KUKA KRL program: EPS_2_26115_SA7007_A_20260219035546.src

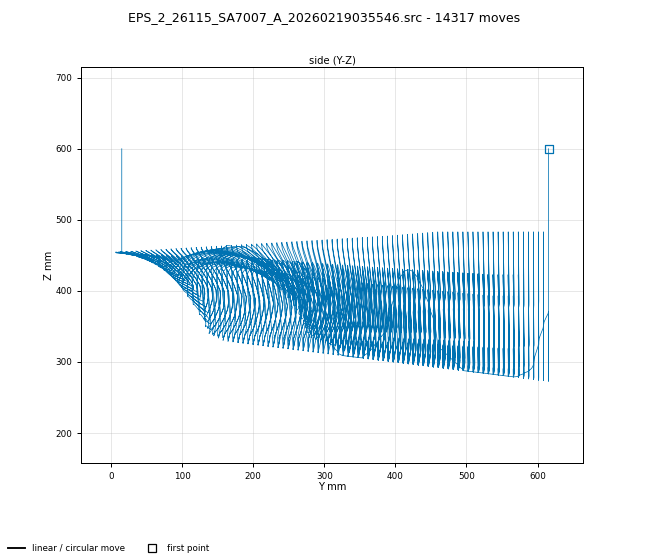
[picture p0: tool path of EPS_2_26115_SA7007_A_20260219035546.src, 14317 of 14319 moves have a stored position in this frame; points joined in program order, loops and branches not executed]
&ACCESS RVP
&REL 4
&COMMENT QRS 19112012
&PARAM EDITMASK = *
DEF PART()
EXT BAS (BAS_COMMAND :IN,REAL :IN )
INT I
BAS (#INITMOV,0 )

;KUKA QRS Post kuka4.cps  Date:22-06-2017 !

File_ID=3063

QRS_PRE_INIT()

;Init var - Until changes are made in qrs_pre_init
Outlet_Square_prg=0
Inlet_1_Square_prg=0
Inlet_2_Square_prg=0
Inlet_3_Square_prg=0
Inlet_4_Square_prg=0
Inlet_5_Square_prg=0

Outlet_1={X 0.000, Y 460.000, Z 382.500, B 0.000, E1 0.000 }
Inlet_1={X 0.000, Y 532.890, Z 292.500, B 0.000, E1 90.000 }
Inlet_2={X 0.000, Y 530.720, Z 322.500, B 0.000, E1 180.000 }
Inlet_3={X 0.000, Y 530.720, Z 322.500, B 0.000, E1 270.000 }
Outlet_1_type=201
Inlet_1_type=201
Inlet_2_type=201
Inlet_3_type=201
;QRS#1=Sidecore dimensions
;QRS#2=200-8" PVC SDR 35 Cut Back
;QRS#3=200-8" PVC SDR 35
;QRS#4=200-8" PVC SDR 35
;QRS#5=200-8" PVC SDR 35
;QRS#6=
;QRS#7=
;QRS#8=
;QRS#9=12-08 PSX
;QRS#10=12-08 PSX
;QRS#11=12-08 PSX
;QRS#12=12-08 PSX
;QRS#13=
;QRS#14=
;QRS#15=
;QRS#16=1220x127x762 2,5'
;QRS#17=EPS Height
;QRS#18=483
;QRS#19=*
;QRS#20= UPDATED VERSION 22-06-2017
;QRS#21=*
Outlet_Square=0100
Inlet_1_Square=0100
Inlet_2_Square=0100
Inlet_3_Square=0100
Inlet_4_Square=0
Inlet_5_Square=0
Mill_Square=1
Outlet_Square_Prg=214
Inlet_1_Square_prg=204
Inlet_2_Square_prg=204
Inlet_3_Square_prg=204

QRS_INIT()

$ADVANCE=5

; T1
PTP {E1 173.498,E2 173.498}
PTP {X 0,Y 615.498,A -85,B 0,C 180,E1 173.498,E2 173.498,E3 0,E4 0,E5 0,E6 0}
QRS_SPEED_INIT()
LIN {X 0,Y 615.498,Z 600,A -85,B 0,C 180,E1 173.498,E2 173.498,E3 0,E4 0,E5 0,E6 0} C_VEL
LIN {X 0,Y 615.498,Z 383.731,A -85,B 0,C 180,E1 173.498,E2 173.498} C_VEL
LIN {X 0,Y 615.498,Z 372.852,A -85,B 0,C 180,E1 173.498,E2 173.498} C_VEL
LIN {X 0,Y 615.496,Z 371.208,A -85,B 0,C 180,E1 173.418,E2 173.418} C_VEL
LIN {X 0,Y 615.497,Z 363.536,A -85,B 0,C 180,E1 172.455,E2 172.455} C_VEL
LIN {X 0,Y 615.498,Z 353.758,A -85,B 0,C 180,E1 171.463,E2 171.463} C_VEL
LIN {X 0,Y 615.498,Z 343.492,A -85,B 0,C 180,E1 170.636,E2 170.636} C_VEL
LIN {X 0,Y 615.458,Z 331.934,A -85,B 0,C 180,E1 169.888,E2 169.888} C_VEL
LIN {X 0,Y 615.433,Z 320.391,A -85,B 0,C 180,E1 169.305,E2 169.305} C_VEL
LIN {X 0,Y 615.457,Z 308.449,A -85,B 0,C 180,E1 168.848,E2 168.848} C_VEL
LIN {X 0,Y 615.487,Z 296.38,A -85,B 0,C 180,E1 168.515,E2 168.515} C_VEL
LIN {X 0,Y 615.495,Z 289.406,A -85,B 0,C 180,E1 168.369,E2 168.369} C_VEL
LIN {X 0,Y 615.472,Z 286.424,A -85,B 0,C 180,E1 166.075,E2 166.075} C_VEL
LIN {X 0,Y 615.45,Z 282.996,A -85,B 0,C 180,E1 163.412,E2 163.412} C_VEL
LIN {X 0,Y 615.494,Z 279.512,A -85,B 0,C 180,E1 160.662,E2 160.662} C_VEL
LIN {X 0,Y 615.46,Z 276.011,A -85,B 0,C 180,E1 157.862,E2 157.862} C_VEL
LIN {X 0,Y 615.467,Z 273.391,A -85,B 0,C 180,E1 155.727,E2 155.727} C_VEL
LIN {X 0,Y 615.489,Z 272.693,A -85,B 0,C 180,E1 155.008,E2 155.008} C_VEL
LIN {X 0,Y 615.468,Z 272.69,A -85,B 0,C 180,E1 152.084,E2 152.084} C_VEL
LIN {X 0,Y 615.473,Z 272.695,A -85,B 0,C 180,E1 149.839,E2 149.839} C_VEL
LIN {X 0,Y 615.495,Z 272.7,A -85,B 0,C 180,E1 147.543,E2 147.543} C_VEL
LIN {X 0,Y 615.482,Z 272.69,A -85,B 0,C 180,E1 145.184,E2 145.184} C_VEL
LIN {X 0,Y 615.492,Z 272.682,A -85,B 0,C 180,E1 142.758,E2 142.758} C_VEL
LIN {X 0,Y 615.496,Z 272.7,A -85,B 0,C 180,E1 139.91,E2 139.91} C_VEL
LIN {X 0,Y 615.488,Z 272.683,A -85,B 0,C 180,E1 136.953,E2 136.953} C_VEL
LIN {X 0,Y 615.489,Z 272.698,A -85,B 0,C 180,E1 133.997,E2 133.997} C_VEL
LIN {X 0,Y 615.487,Z 272.684,A -85,B 0,C 180,E1 131.094,E2 131.094} C_VEL
LIN {X 0,Y 615.488,Z 272.687,A -85,B 0,C 180,E1 128.905,E2 128.905} C_VEL
LIN {X 0,Y 615.484,Z 272.704,A -85,B 0,C 180,E1 126.425,E2 126.425} C_VEL
LIN {X 0,Y 615.49,Z 272.727,A -85,B 0,C 180,E1 124.701,E2 124.701} C_VEL
LIN {X 0,Y 615.482,Z 277.506,A -85,B 0,C 180,E1 122.329,E2 122.329} C_VEL
LIN {X 0,Y 615.472,Z 282.453,A -85,B 0,C 180,E1 119.791,E2 119.791} C_VEL
LIN {X 0,Y 615.46,Z 287.533,A -85,B 0,C 180,E1 117.039,E2 117.039} C_VEL
LIN {X 0,Y 615.461,Z 291.397,A -85,B 0,C 180,E1 114.993,E2 114.993} C_VEL
LIN {X 0,Y 615.482,Z 296.491,A -85,B 0,C 180,E1 112.344,E2 112.344} C_VEL
LIN {X 0,Y 615.482,Z 301.009,A -85,B 0,C 180,E1 110.033,E2 110.033} C_VEL
LIN {X 0,Y 615.484,Z 306.513,A -85,B 0,C 180,E1 107.271,E2 107.271} C_VEL
LIN {X 0,Y 615.467,Z 311.996,A -85,B 0,C 180,E1 104.55,E2 104.55} C_VEL
LIN {X 0,Y 615.479,Z 317.495,A -85,B 0,C 180,E1 101.861,E2 101.861} C_VEL
LIN {X 0,Y 615.496,Z 318.09,A -85,B 0,C 180,E1 101.568,E2 101.568} C_VEL
LIN {X 0,Y 615.485,Z 332.738,A -85,B 0,C 180,E1 101.235,E2 101.235} C_VEL
LIN {X 0,Y 615.452,Z 345.032,A -85,B 0,C 180,E1 100.827,E2 100.827} C_VEL
LIN {X 0,Y 615.452,Z 357.201,A -85,B 0,C 180,E1 100.278,E2 100.278} C_VEL
LIN {X 0,Y 615.496,Z 368.575,A -85,B 0,C 180,E1 99.613,E2 99.613} C_VEL
LIN {X 0,Y 615.498,Z 378.822,A -85,B 0,C 180,E1 98.867,E2 98.867} C_VEL
LIN {X 0,Y 615.498,Z 388.033,A -85,B 0,C 180,E1 98.041,E2 98.041} C_VEL
LIN {X 0,Y 615.499,Z 396.892,A -85,B 0,C 180,E1 97.057,E2 97.057} C_VEL
LIN {X 0,Y 615.497,Z 404.123,A -85,B 0,C 180,E1 96.063,E2 96.063} C_VEL
LIN {X 0,Y 615.497,Z 408.958,A -85,B 0,C 180,E1 95.241,E2 95.241} C_VEL
LIN {X 0,Y 615.494,Z 413.658,A -85,B 0,C 180,E1 94.256,E2 94.256} C_VEL
LIN {X 0,Y 615.494,Z 417.254,A -85,B 0,C 180,E1 93.273,E2 93.273} C_VEL
LIN {X 0,Y 615.496,Z 419.115,A -85,B 0,C 180,E1 92.618,E2 92.618} C_VEL
LIN {X 0,Y 615.5,Z 420.533,A -85,B 0,C 180,E1 91.963,E2 91.963} C_VEL
LIN {X 0,Y 615.496,Z 422.141,A -85,B 0,C 180,E1 90.654,E2 90.654} C_VEL
LIN {X 0,Y 615.495,Z 422.384,A -85,B 0,C 180,E1 90,E2 90} C_VEL
LIN {X 0,Y 615.495,Z 422.206,A -85,B 0,C 180,E1 89.346,E2 89.346} C_VEL
LIN {X 0,Y 615.5,Z 420.682,A -85,B 0,C 180,E1 88.037,E2 88.037} C_VEL
LIN {X 0,Y 615.498,Z 419.341,A -85,B 0,C 180,E1 87.382,E2 87.382} C_VEL
LIN {X 0,Y 615.496,Z 416.494,A -85,B 0,C 180,E1 86.399,E2 86.399} C_VEL
LIN {X 0,Y 615.498,Z 412.634,A -85,B 0,C 180,E1 85.416,E2 85.416} C_VEL
LIN {X 0,Y 615.498,Z 407.651,A -85,B 0,C 180,E1 84.43,E2 84.43} C_VEL
LIN {X 0,Y 615.496,Z 401.208,A -85,B 0,C 180,E1 83.418,E2 83.418} C_VEL
LIN {X 0,Y 615.497,Z 393.536,A -85,B 0,C 180,E1 82.455,E2 82.455} C_VEL
LIN {X 0,Y 615.498,Z 383.758,A -85,B 0,C 180,E1 81.463,E2 81.463} C_VEL
LIN {X 0,Y 615.498,Z 373.492,A -85,B 0,C 180,E1 80.636,E2 80.636} C_VEL
LIN {X 0,Y 615.46,Z 361.934,A -85,B 0,C 180,E1 79.888,E2 79.888} C_VEL
LIN {X 0,Y 615.439,Z 350.346,A -85,B 0,C 180,E1 79.303,E2 79.303} C_VEL
LIN {X 0,Y 615.467,Z 338.434,A -85,B 0,C 180,E1 78.848,E2 78.848} C_VEL
LIN {X 0,Y 615.494,Z 326.38,A -85,B 0,C 180,E1 78.515,E2 78.515} C_VEL
LIN {X 0,Y 615.497,Z 318.103,A -85,B 0,C 180,E1 78.348,E2 78.348} C_VEL
LIN {X 0,Y 615.476,Z 313.45,A -85,B 0,C 180,E1 76.073,E2 76.073} C_VEL
LIN {X 0,Y 615.476,Z 308.058,A -85,B 0,C 180,E1 73.413,E2 73.413} C_VEL
LIN {X 0,Y 615.486,Z 302.567,A -85,B 0,C 180,E1 70.662,E2 70.662} C_VEL
LIN {X 0,Y 615.487,Z 297.064,A -85,B 0,C 180,E1 67.863,E2 67.863} C_VEL
LIN {X 0,Y 615.483,Z 292.945,A -85,B 0,C 180,E1 65.728,E2 65.728} C_VEL
LIN {X 0,Y 615.456,Z 288.826,A -85,B 0,C 180,E1 63.554,E2 63.554} C_VEL
LIN {X 0,Y 615.441,Z 284.694,A -85,B 0,C 180,E1 61.339,E2 61.339} C_VEL
LIN {X 0,Y 615.495,Z 280.115,A -85,B 0,C 180,E1 58.913,E2 58.913} C_VEL
LIN {X 0,Y 615.481,Z 275.287,A -85,B 0,C 180,E1 56.467,E2 56.467} C_VEL
LIN {X 0,Y 615.491,Z 272.697,A -85,B 0,C 180,E1 55.185,E2 55.185} C_VEL
LIN {X 0,Y 615.489,Z 272.701,A -85,B 0,C 180,E1 52.758,E2 52.758} C_VEL
LIN {X 0,Y 615.472,Z 272.7,A -85,B 0,C 180,E1 49.913,E2 49.913} C_VEL
LIN {X 0,Y 615.492,Z 272.693,A -85,B 0,C 180,E1 46.953,E2 46.953} C_VEL
LIN {X 0,Y 615.466,Z 272.7,A -85,B 0,C 180,E1 44.152,E2 44.152} C_VEL
LIN {X 0,Y 615.469,Z 272.7,A -85,B 0,C 180,E1 41.476,E2 41.476} C_VEL
LIN {X 0,Y 615.492,Z 272.694,A -85,B 0,C 180,E1 38.904,E2 38.904} C_VEL
LIN {X 0,Y 615.464,Z 272.7,A -85,B 0,C 180,E1 36.427,E2 36.427} C_VEL
LIN {X 0,Y 615.489,Z 272.727,A -85,B 0,C 180,E1 34.815,E2 34.815} C_VEL
LIN {X 0,Y 615.484,Z 277.586,A -85,B 0,C 180,E1 32.33,E2 32.33} C_VEL
LIN {X 0,Y 615.471,Z 282.454,A -85,B 0,C 180,E1 29.791,E2 29.791} C_VEL
LIN {X 0,Y 615.459,Z 287.533,A -85,B 0,C 180,E1 27.039,E2 27.039} C_VEL
LIN {X 0,Y 615.461,Z 291.397,A -85,B 0,C 180,E1 24.993,E2 24.993} C_VEL
LIN {X 0,Y 615.482,Z 296.491,A -85,B 0,C 180,E1 22.344,E2 22.344} C_VEL
LIN {X 0,Y 615.482,Z 301.009,A -85,B 0,C 180,E1 20.033,E2 20.033} C_VEL
LIN {X 0,Y 615.485,Z 306.513,A -85,B 0,C 180,E1 17.271,E2 17.271} C_VEL
LIN {X 0,Y 615.468,Z 311.996,A -85,B 0,C 180,E1 14.55,E2 14.55} C_VEL
LIN {X 0,Y 615.479,Z 317.495,A -85,B 0,C 180,E1 11.861,E2 11.861} C_VEL
LIN {X 0,Y 615.496,Z 318.09,A -85,B 0,C 180,E1 11.568,E2 11.568} C_VEL
LIN {X 0,Y 615.485,Z 332.737,A -85,B 0,C 180,E1 11.235,E2 11.235} C_VEL
LIN {X 0,Y 615.452,Z 345.032,A -85,B 0,C 180,E1 10.827,E2 10.827} C_VEL
LIN {X 0,Y 615.452,Z 357.2,A -85,B 0,C 180,E1 10.278,E2 10.278} C_VEL
LIN {X 0,Y 615.496,Z 368.574,A -85,B 0,C 180,E1 9.613,E2 9.613} C_VEL
LIN {X 0,Y 615.498,Z 378.822,A -85,B 0,C 180,E1 8.867,E2 8.867} C_VEL
LIN {X 0,Y 615.498,Z 388.033,A -85,B 0,C 180,E1 8.041,E2 8.041} C_VEL
LIN {X 0,Y 615.499,Z 396.891,A -85,B 0,C 180,E1 7.057,E2 7.057} C_VEL
LIN {X 0,Y 615.497,Z 404.123,A -85,B 0,C 180,E1 6.063,E2 6.063} C_VEL
LIN {X 0,Y 615.497,Z 408.958,A -85,B 0,C 180,E1 5.241,E2 5.241} C_VEL
LIN {X 0,Y 615.494,Z 413.658,A -85,B 0,C 180,E1 4.256,E2 4.256} C_VEL
LIN {X 0,Y 615.494,Z 417.254,A -85,B 0,C 180,E1 3.273,E2 3.273} C_VEL
LIN {X 0,Y 615.496,Z 419.115,A -85,B 0,C 180,E1 2.618,E2 2.618} C_VEL
LIN {X 0,Y 615.5,Z 420.533,A -85,B 0,C 180,E1 1.963,E2 1.963} C_VEL
LIN {X 0,Y 615.496,Z 422.141,A -85,B 0,C 180,E1 0.654,E2 0.654} C_VEL
LIN {X 0,Y 615.495,Z 422.384,A -85,B 0,C 180,E1 0,E2 0} C_VEL
LIN {X 0,Y 615.495,Z 422.206,A -85,B 0,C 180,E1 -0.654,E2 -0.654} C_VEL
LIN {X 0,Y 615.5,Z 420.682,A -85,B 0,C 180,E1 -1.963,E2 -1.963} C_VEL
LIN {X 0,Y 615.498,Z 419.341,A -85,B 0,C 180,E1 -2.618,E2 -2.618} C_VEL
LIN {X 0,Y 615.496,Z 416.494,A -85,B 0,C 180,E1 -3.601,E2 -3.601} C_VEL
LIN {X 0,Y 615.498,Z 412.634,A -85,B 0,C 180,E1 -4.584,E2 -4.584} C_VEL
LIN {X 0,Y 615.498,Z 407.651,A -85,B 0,C 180,E1 -5.57,E2 -5.57} C_VEL
LIN {X 0,Y 615.496,Z 401.208,A -85,B 0,C 180,E1 -6.582,E2 -6.582} C_VEL
LIN {X 0,Y 615.497,Z 393.537,A -85,B 0,C 180,E1 -7.545,E2 -7.545} C_VEL
LIN {X 0,Y 615.498,Z 383.759,A -85,B 0,C 180,E1 -8.536,E2 -8.536} C_VEL
LIN {X 0,Y 615.498,Z 373.493,A -85,B 0,C 180,E1 -9.364,E2 -9.364} C_VEL
LIN {X 0,Y 615.46,Z 361.935,A -85,B 0,C 180,E1 -10.112,E2 -10.112} C_VEL
LIN {X 0,Y 615.439,Z 350.346,A -85,B 0,C 180,E1 -10.697,E2 -10.697} C_VEL
LIN {X 0,Y 615.467,Z 338.435,A -85,B 0,C 180,E1 -11.152,E2 -11.152} C_VEL
LIN {X 0,Y 615.494,Z 326.382,A -85,B 0,C 180,E1 -11.485,E2 -11.485} C_VEL
LIN {X 0,Y 615.497,Z 318.103,A -85,B 0,C 180,E1 -11.652,E2 -11.652} C_VEL
LIN {X 0,Y 615.476,Z 313.45,A -85,B 0,C 180,E1 -13.927,E2 -13.927} C_VEL
LIN {X 0,Y 615.476,Z 308.058,A -85,B 0,C 180,E1 -16.587,E2 -16.587} C_VEL
LIN {X 0,Y 615.486,Z 302.567,A -85,B 0,C 180,E1 -19.338,E2 -19.338} C_VEL
LIN {X 0,Y 615.487,Z 297.064,A -85,B 0,C 180,E1 -22.137,E2 -22.137} C_VEL
LIN {X 0,Y 615.483,Z 292.945,A -85,B 0,C 180,E1 -24.272,E2 -24.272} C_VEL
LIN {X 0,Y 615.456,Z 288.826,A -85,B 0,C 180,E1 -26.446,E2 -26.446} C_VEL
LIN {X 0,Y 615.441,Z 284.694,A -85,B 0,C 180,E1 -28.66,E2 -28.66} C_VEL
LIN {X 0,Y 615.495,Z 280.243,A -85,B 0,C 180,E1 -30.919,E2 -30.919} C_VEL
LIN {X 0,Y 615.493,Z 274.102,A -85,B 0,C 180,E1 -33.534,E2 -33.534} C_VEL
LIN {X 0,Y 615.472,Z 272.7,A -85,B 0,C 180,E1 -34.107,E2 -34.107} C_VEL
LIN {X 0,Y 615.489,Z 272.694,A -85,B 0,C 180,E1 -36.936,E2 -36.936} C_VEL
LIN {X 0,Y 615.463,Z 272.699,A -85,B 0,C 180,E1 -39.752,E2 -39.752} C_VEL
LIN {X 0,Y 615.46,Z 272.7,A -85,B 0,C 180,E1 -42.356,E2 -42.356} C_VEL
LIN {X 0,Y 615.493,Z 272.693,A -85,B 0,C 180,E1 -45.068,E2 -45.068} C_VEL
LIN {X 0,Y 615.467,Z 272.7,A -85,B 0,C 180,E1 -47.922,E2 -47.922} C_VEL
LIN {X 0,Y 615.461,Z 272.7,A -85,B 0,C 180,E1 -50.248,E2 -50.248} C_VEL
LIN {X 0,Y 615.49,Z 272.694,A -85,B 0,C 180,E1 -53.063,E2 -53.063} C_VEL
LIN {X 0,Y 615.469,Z 272.843,A -85,B 0,C 180,E1 -54.483,E2 -54.483} C_VEL
LIN {X 0,Y 615.449,Z 283.202,A -85,B 0,C 180,E1 -57.151,E2 -57.151} C_VEL
LIN {X 0,Y 615.438,Z 292.407,A -85,B 0,C 180,E1 -59.458,E2 -59.458} C_VEL
LIN {X 0,Y 615.482,Z 303.134,A -85,B 0,C 180,E1 -62.084,E2 -62.084} C_VEL
LIN {X 0,Y 615.484,Z 314.169,A -85,B 0,C 180,E1 -64.72,E2 -64.72} C_VEL
LIN {X 0,Y 615.48,Z 325.649,A -85,B 0,C 180,E1 -67.405,E2 -67.405} C_VEL
LIN {X 0,Y 615.477,Z 336.812,A -85,B 0,C 180,E1 -69.967,E2 -69.967} C_VEL
LIN {X 0,Y 615.487,Z 349.039,A -85,B 0,C 180,E1 -72.729,E2 -72.729} C_VEL
LIN {X 0,Y 615.461,Z 361.262,A -85,B 0,C 180,E1 -75.45,E2 -75.45} C_VEL
LIN {X 0,Y 615.478,Z 373.471,A -85,B 0,C 180,E1 -78.139,E2 -78.139} C_VEL
LIN {X 0,Y 615.498,Z 374.458,A -85,B 0,C 180,E1 -78.348,E2 -78.348} C_VEL
LIN {X 0,Y 615.499,Z 388.06,A -85,B 0,C 180,E1 -78.599,E2 -78.599} C_VEL
LIN {X 0,Y 615.459,Z 400.775,A -85,B 0,C 180,E1 -78.969,E2 -78.969} C_VEL
LIN {X 0,Y 615.441,Z 413.029,A -85,B 0,C 180,E1 -79.472,E2 -79.472} C_VEL
LIN {X 0,Y 615.479,Z 423.982,A -85,B 0,C 180,E1 -80.055,E2 -80.055} C_VEL
LIN {X 0,Y 615.499,Z 435.167,A -85,B 0,C 180,E1 -80.801,E2 -80.801} C_VEL
LIN {X 0,Y 615.498,Z 445.044,A -85,B 0,C 180,E1 -81.629,E2 -81.629} C_VEL
LIN {X 0,Y 615.498,Z 454.606,A -85,B 0,C 180,E1 -82.62,E2 -82.62} C_VEL
LIN {X 0,Y 615.496,Z 462.203,A -85,B 0,C 180,E1 -83.608,E2 -83.608} C_VEL
LIN {X 0,Y 615.498,Z 469.204,A -85,B 0,C 180,E1 -84.759,E2 -84.759} C_VEL
LIN {X 0,Y 615.494,Z 473.851,A -85,B 0,C 180,E1 -85.744,E2 -85.744} C_VEL
LIN {X 0,Y 615.494,Z 477.399,A -85,B 0,C 180,E1 -86.727,E2 -86.727} C_VEL
LIN {X 0,Y 615.497,Z 479.233,A -85,B 0,C 180,E1 -87.382,E2 -87.382} C_VEL
LIN {X 0,Y 615.5,Z 480.607,A -85,B 0,C 180,E1 -88.037,E2 -88.037} C_VEL
LIN {X 0,Y 615.496,Z 482.173,A -85,B 0,C 180,E1 -89.346,E2 -89.346} C_VEL
LIN {X 0,Y 615.494,Z 482.389,A -85,B 0,C 180,E1 -90,E2 -90} C_VEL
LIN {X 0,Y 615.495,Z 481.58,A -85,B 0,C 180,E1 -91.309,E2 -91.309} C_VEL
LIN {X 0,Y 615.5,Z 480.607,A -85,B 0,C 180,E1 -91.963,E2 -91.963} C_VEL
LIN {X 0,Y 615.497,Z 479.233,A -85,B 0,C 180,E1 -92.618,E2 -92.618} C_VEL
LIN {X 0,Y 615.496,Z 476.349,A -85,B 0,C 180,E1 -93.601,E2 -93.601} C_VEL
LIN {X 0,Y 615.498,Z 472.441,A -85,B 0,C 180,E1 -94.584,E2 -94.584} C_VEL
LIN {X 0,Y 615.499,Z 467.405,A -85,B 0,C 180,E1 -95.57,E2 -95.57} C_VEL
LIN {X 0,Y 615.497,Z 460.869,A -85,B 0,C 180,E1 -96.583,E2 -96.583} C_VEL
LIN {X 0,Y 615.497,Z 453.133,A -85,B 0,C 180,E1 -97.545,E2 -97.545} C_VEL
LIN {X 0,Y 615.498,Z 445.044,A -85,B 0,C 180,E1 -98.371,E2 -98.371} C_VEL
LIN {X 0,Y 615.499,Z 435.167,A -85,B 0,C 180,E1 -99.199,E2 -99.199} C_VEL
LIN {X 0,Y 615.479,Z 423.982,A -85,B 0,C 180,E1 -99.945,E2 -99.945} C_VEL
LIN {X 0,Y 615.441,Z 413.029,A -85,B 0,C 180,E1 -100.528,E2 -100.528} C_VEL
LIN {X 0,Y 615.459,Z 400.775,A -85,B 0,C 180,E1 -101.031,E2 -101.031} C_VEL
LIN {X 0,Y 615.499,Z 388.06,A -85,B 0,C 180,E1 -101.401,E2 -101.401} C_VEL
LIN {X 0,Y 615.498,Z 374.323,A -85,B 0,C 180,E1 -101.673,E2 -101.673} C_VEL
LIN {X 0,Y 615.46,Z 362.674,A -85,B 0,C 180,E1 -104.239,E2 -104.239} C_VEL
LIN {X 0,Y 615.491,Z 350.564,A -85,B 0,C 180,E1 -106.928,E2 -106.928} C_VEL
LIN {X 0,Y 615.487,Z 338.344,A -85,B 0,C 180,E1 -109.685,E2 -109.685} C_VEL
LIN {X 0,Y 615.491,Z 326.724,A -85,B 0,C 180,E1 -112.346,E2 -112.346} C_VEL
LIN {X 0,Y 615.467,Z 315.393,A -85,B 0,C 180,E1 -114.993,E2 -114.993} C_VEL
LIN {X 0,Y 615.496,Z 304.666,A -85,B 0,C 180,E1 -117.545,E2 -117.545} C_VEL
LIN {X 0,Y 615.448,Z 293.939,A -85,B 0,C 180,E1 -120.162,E2 -120.162} C_VEL
LIN {X 0,Y 615.429,Z 284.737,A -85,B 0,C 180,E1 -122.461,E2 -122.461} C_VEL
LIN {X 0,Y 615.493,Z 273.994,A -85,B 0,C 180,E1 -125.214,E2 -125.214} C_VEL
LIN {X 0,Y 615.447,Z 272.698,A -85,B 0,C 180,E1 -125.619,E2 -125.619} C_VEL
LIN {X 0,Y 615.425,Z 272.698,A -85,B 0,C 180,E1 -128.073,E2 -128.073} C_VEL
LIN {X 0,Y 615.433,Z 272.697,A -85,B 0,C 180,E1 -130.083,E2 -130.083} C_VEL
LIN {X 0,Y 615.458,Z 272.698,A -85,B 0,C 180,E1 -132.356,E2 -132.356} C_VEL
LIN {X 0,Y 615.491,Z 272.688,A -85,B 0,C 180,E1 -135.068,E2 -135.068} C_VEL
LIN {X 0,Y 615.453,Z 272.693,A -85,B 0,C 180,E1 -137.644,E2 -137.644} C_VEL
LIN {X 0,Y 615.497,Z 272.7,A -85,B 0,C 180,E1 -140.25,E2 -140.25} C_VEL
LIN {X 0,Y 615.478,Z 272.686,A -85,B 0,C 180,E1 -143.065,E2 -143.065} C_VEL
LIN {X 0,Y 615.496,Z 272.699,A -85,B 0,C 180,E1 -145.978,E2 -145.978} C_VEL
LIN {X 0,Y 615.484,Z 272.685,A -85,B 0,C 180,E1 -148.915,E2 -148.915} C_VEL
LIN {X 0,Y 615.496,Z 272.699,A -85,B 0,C 180,E1 -151.549,E2 -151.549} C_VEL
LIN {X 0,Y 615.484,Z 272.685,A -85,B 0,C 180,E1 -154.432,E2 -154.432} C_VEL
LIN {X 0,Y 615.485,Z 272.692,A -85,B 0,C 180,E1 -155.008,E2 -155.008} C_VEL
LIN {X 0,Y 615.485,Z 274.153,A -85,B 0,C 180,E1 -156.443,E2 -156.443} C_VEL
LIN {X 0,Y 615.473,Z 277.868,A -85,B 0,C 180,E1 -159.447,E2 -159.447} C_VEL
LIN {X 0,Y 615.467,Z 281.135,A -85,B 0,C 180,E1 -162.042,E2 -162.042} C_VEL
LIN {X 0,Y 615.494,Z 284.626,A -85,B 0,C 180,E1 -164.774,E2 -164.774} C_VEL
LIN {X 0,Y 615.444,Z 288.115,A -85,B 0,C 180,E1 -167.469,E2 -167.469} C_VEL
LIN {X 0,Y 615.496,Z 289.398,A -85,B 0,C 180,E1 -168.453,E2 -168.453} C_VEL
LIN {X 0,Y 615.473,Z 304.258,A -85,B 0,C 180,E1 -168.807,E2 -168.807} C_VEL
LIN {X 0,Y 615.443,Z 316.21,A -85,B 0,C 180,E1 -169.218,E2 -169.218} C_VEL
LIN {X 0,Y 615.454,Z 328.762,A -85,B 0,C 180,E1 -169.805,E2 -169.805} C_VEL
LIN {X 0,Y 615.499,Z 339.847,A -85,B 0,C 180,E1 -170.47,E2 -170.47} C_VEL
LIN {X 0,Y 615.498,Z 348.822,A -85,B 0,C 180,E1 -171.133,E2 -171.133} C_VEL
LIN {X 0,Y 615.498,Z 358.034,A -85,B 0,C 180,E1 -171.959,E2 -171.959} C_VEL
LIN {X 0,Y 615.499,Z 366.892,A -85,B 0,C 180,E1 -172.943,E2 -172.943} C_VEL
LIN {X 0,Y 615.497,Z 374.123,A -85,B 0,C 180,E1 -173.937,E2 -173.937} C_VEL
LIN {X 0,Y 615.497,Z 378.958,A -85,B 0,C 180,E1 -174.759,E2 -174.759} C_VEL
LIN {X 0,Y 615.494,Z 383.658,A -85,B 0,C 180,E1 -175.744,E2 -175.744} C_VEL
LIN {X 0,Y 615.494,Z 387.255,A -85,B 0,C 180,E1 -176.727,E2 -176.727} C_VEL
LIN {X 0,Y 615.496,Z 389.115,A -85,B 0,C 180,E1 -177.382,E2 -177.382} C_VEL
LIN {X 0,Y 615.5,Z 390.533,A -85,B 0,C 180,E1 -178.037,E2 -178.037} C_VEL
LIN {X 0,Y 615.496,Z 392.142,A -85,B 0,C 180,E1 -179.346,E2 -179.346} C_VEL
LIN {X 0,Y 615.495,Z 392.384,A -85,B 0,C 180,E1 -180,E2 -180} C_VEL
LIN {X 0,Y 615.495,Z 392.206,A -85,B 0,C 180,E1 -180.654,E2 -180.654} C_VEL
LIN {X 0,Y 615.5,Z 390.682,A -85,B 0,C 180,E1 -181.963,E2 -181.963} C_VEL
LIN {X 0,Y 615.498,Z 389.341,A -85,B 0,C 180,E1 -182.618,E2 -182.618} C_VEL
LIN {X 0,Y 615.496,Z 386.494,A -85,B 0,C 180,E1 -183.601,E2 -183.601} C_VEL
LIN {X 0,Y 615.498,Z 382.634,A -85,B 0,C 180,E1 -184.585,E2 -184.585} C_VEL
LIN {X 0,Y 615.498,Z 377.651,A -85,B 0,C 180,E1 -185.57,E2 -185.57} C_VEL
LIN {X 0,Y 615.496,Z 371.208,A -85,B 0,C 180,E1 -186.582,E2 -186.582} C_VEL
LIN {X 0,Y 614.829,Z 368.026,A -85,B 0,C 180,E1 -187.031,E2 -187.031} C_VEL
LIN {X 0,Y 611.989,Z 362.453,A -85,B 0,C 180,E1 -187.748,E2 -187.748} C_VEL
LIN {X 0,Y 609.138,Z 356.178,A -85,B 0,C 180,E1 -188.429,E2 -188.429} C_VEL
LIN {X 0,Y 608.477,Z 351.937,A -85,B 0,C 180,E1 -188.819,E2 -188.819} C_VEL
LIN {X 0,Y 608.496,Z 341.391,A -85,B 0,C 180,E1 -189.641,E2 -189.641} C_VEL
LIN {X 0,Y 608.448,Z 330.608,A -85,B 0,C 180,E1 -190.314,E2 -190.314} C_VEL
LIN {X 0,Y 608.45,Z 318.725,A -85,B 0,C 180,E1 -190.896,E2 -190.896} C_VEL
LIN {X 0,Y 608.514,Z 305.969,A -85,B 0,C 180,E1 -191.365,E2 -191.365} C_VEL
LIN {X 0,Y 608.557,Z 293.642,A -85,B 0,C 180,E1 -191.681,E2 -191.681} C_VEL
LIN {X 0,Y 608.436,Z 289.897,A -85,B 0,C 180,E1 -191.768,E2 -191.768} C_VEL
LIN {X 0,Y 608.405,Z 286.957,A -85,B 0,C 180,E1 -194.039,E2 -194.039} C_VEL
LIN {X 0,Y 608.4,Z 283.44,A -85,B 0,C 180,E1 -196.786,E2 -196.786} C_VEL
LIN {X 0,Y 608.409,Z 279.922,A -85,B 0,C 180,E1 -199.572,E2 -199.572} C_VEL
LIN {X 0,Y 608.402,Z 276.338,A -85,B 0,C 180,E1 -202.462,E2 -202.462} C_VEL
LIN {X 0,Y 608.415,Z 273.766,A -85,B 0,C 180,E1 -204.573,E2 -204.573} C_VEL
LIN {X 0,Y 608.481,Z 273.686,A -85,B 0,C 180,E1 -207.207,E2 -207.207} C_VEL
LIN {X 0,Y 608.454,Z 273.69,A -85,B 0,C 180,E1 -209.969,E2 -209.969} C_VEL
LIN {X 0,Y 608.462,Z 273.689,A -85,B 0,C 180,E1 -212.879,E2 -212.879} C_VEL
LIN {X 0,Y 608.437,Z 273.69,A -85,B 0,C 180,E1 -215.278,E2 -215.278} C_VEL
LIN {X 0,Y 608.472,Z 273.689,A -85,B 0,C 180,E1 -217.746,E2 -217.746} C_VEL
LIN {X 0,Y 608.453,Z 273.694,A -85,B 0,C 180,E1 -220.329,E2 -220.329} C_VEL
LIN {X 0,Y 608.454,Z 273.688,A -85,B 0,C 180,E1 -222.96,E2 -222.96} C_VEL
LIN {X 0,Y 608.465,Z 273.694,A -85,B 0,C 180,E1 -225.736,E2 -225.736} C_VEL
LIN {X 0,Y 608.457,Z 273.687,A -85,B 0,C 180,E1 -228.659,E2 -228.659} C_VEL
LIN {X 0,Y 608.462,Z 273.695,A -85,B 0,C 180,E1 -231.761,E2 -231.761} C_VEL
LIN {X 0,Y 608.443,Z 273.693,A -85,B 0,C 180,E1 -233.955,E2 -233.955} C_VEL
LIN {X 0,Y 608.434,Z 273.868,A -85,B 0,C 180,E1 -235.42,E2 -235.42} C_VEL
LIN {X 0,Y 608.427,Z 278.82,A -85,B 0,C 180,E1 -237.903,E2 -237.903} C_VEL
LIN {X 0,Y 608.422,Z 283.309,A -85,B 0,C 180,E1 -240.218,E2 -240.218} C_VEL
LIN {X 0,Y 608.397,Z 288.889,A -85,B 0,C 180,E1 -243.223,E2 -243.223} C_VEL
LIN {X 0,Y 608.409,Z 293.036,A -85,B 0,C 180,E1 -245.427,E2 -245.427} C_VEL
LIN {X 0,Y 608.449,Z 298.565,A -85,B 0,C 180,E1 -248.308,E2 -248.308} C_VEL
LIN {X 0,Y 608.429,Z 304.425,A -85,B 0,C 180,E1 -251.297,E2 -251.297} C_VEL
LIN {X 0,Y 608.437,Z 309.624,A -85,B 0,C 180,E1 -253.905,E2 -253.905} C_VEL
LIN {X 0,Y 608.434,Z 315.154,A -85,B 0,C 180,E1 -256.643,E2 -256.643} C_VEL
LIN {X 0,Y 608.455,Z 318.773,A -85,B 0,C 180,E1 -258.317,E2 -258.317} C_VEL
LIN {X 0,Y 608.538,Z 332.12,A -85,B 0,C 180,E1 -258.614,E2 -258.614} C_VEL
LIN {X 0,Y 608.473,Z 345.103,A -85,B 0,C 180,E1 -259.044,E2 -259.044} C_VEL
LIN {X 0,Y 608.459,Z 357.365,A -85,B 0,C 180,E1 -259.602,E2 -259.602} C_VEL
LIN {X 0,Y 608.505,Z 368.789,A -85,B 0,C 180,E1 -260.275,E2 -260.275} C_VEL
LIN {X 0,Y 608.474,Z 379.084,A -85,B 0,C 180,E1 -261.029,E2 -261.029} C_VEL
LIN {X 0,Y 608.464,Z 388.346,A -85,B 0,C 180,E1 -261.866,E2 -261.866} C_VEL
LIN {X 0,Y 608.466,Z 397.32,A -85,B 0,C 180,E1 -262.867,E2 -262.867} C_VEL
LIN {X 0,Y 608.444,Z 404.555,A -85,B 0,C 180,E1 -263.867,E2 -263.867} C_VEL
LIN {X 0,Y 608.462,Z 409.434,A -85,B 0,C 180,E1 -264.698,E2 -264.698} C_VEL
LIN {X 0,Y 608.439,Z 414.179,A -85,B 0,C 180,E1 -265.694,E2 -265.694} C_VEL
LIN {X 0,Y 608.425,Z 417.813,A -85,B 0,C 180,E1 -266.689,E2 -266.689} C_VEL
LIN {X 0,Y 608.425,Z 419.689,A -85,B 0,C 180,E1 -267.352,E2 -267.352} C_VEL
LIN {X 0,Y 608.445,Z 421.126,A -85,B 0,C 180,E1 -268.014,E2 -268.014} C_VEL
LIN {X 0,Y 608.439,Z 422.752,A -85,B 0,C 180,E1 -269.338,E2 -269.338} C_VEL
LIN {X 0,Y 608.435,Z 422.995,A -85,B 0,C 180,E1 -270,E2 -270} C_VEL
LIN {X 0,Y 608.438,Z 422.815,A -85,B 0,C 180,E1 -270.662,E2 -270.662} C_VEL
LIN {X 0,Y 608.445,Z 421.276,A -85,B 0,C 180,E1 -271.986,E2 -271.986} C_VEL
LIN {X 0,Y 608.426,Z 419.919,A -85,B 0,C 180,E1 -272.648,E2 -272.648} C_VEL
LIN {X 0,Y 608.449,Z 417.042,A -85,B 0,C 180,E1 -273.642,E2 -273.642} C_VEL
LIN {X 0,Y 608.433,Z 413.143,A -85,B 0,C 180,E1 -274.638,E2 -274.638} C_VEL
LIN {X 0,Y 608.45,Z 408.112,A -85,B 0,C 180,E1 -275.634,E2 -275.634} C_VEL
LIN {X 0,Y 608.441,Z 401.792,A -85,B 0,C 180,E1 -276.633,E2 -276.633} C_VEL
LIN {X 0,Y 608.475,Z 393.879,A -85,B 0,C 180,E1 -277.633,E2 -277.633} C_VEL
LIN {X 0,Y 608.472,Z 384.035,A -85,B 0,C 180,E1 -278.636,E2 -278.636} C_VEL
LIN {X 0,Y 608.481,Z 373.711,A -85,B 0,C 180,E1 -279.473,E2 -279.473} C_VEL
LIN {X 0,Y 608.472,Z 362.098,A -85,B 0,C 180,E1 -280.229,E2 -280.229} C_VEL
LIN {X 0,Y 608.465,Z 350.462,A -85,B 0,C 180,E1 -280.821,E2 -280.821} C_VEL
LIN {X 0,Y 608.496,Z 338.407,A -85,B 0,C 180,E1 -281.286,E2 -281.286} C_VEL
LIN {X 0,Y 608.537,Z 325.549,A -85,B 0,C 180,E1 -281.639,E2 -281.639} C_VEL
LIN {X 0,Y 608.441,Z 318.536,A -85,B 0,C 180,E1 -281.789,E2 -281.789} C_VEL
LIN {X 0,Y 608.428,Z 313.954,A -85,B 0,C 180,E1 -284.038,E2 -284.038} C_VEL
LIN {X 0,Y 608.411,Z 308.422,A -85,B 0,C 180,E1 -286.785,E2 -286.785} C_VEL
LIN {X 0,Y 608.431,Z 302.89,A -85,B 0,C 180,E1 -289.571,E2 -289.571} C_VEL
LIN {X 0,Y 608.432,Z 297.237,A -85,B 0,C 180,E1 -292.469,E2 -292.469} C_VEL
LIN {X 0,Y 608.414,Z 293.207,A -85,B 0,C 180,E1 -294.573,E2 -294.573} C_VEL
LIN {X 0,Y 608.426,Z 288.272,A -85,B 0,C 180,E1 -297.197,E2 -297.197} C_VEL
LIN {X 0,Y 608.439,Z 283.112,A -85,B 0,C 180,E1 -299.966,E2 -299.966} C_VEL
LIN {X 0,Y 608.431,Z 278.17,A -85,B 0,C 180,E1 -302.517,E2 -302.517} C_VEL
LIN {X 0,Y 608.486,Z 273.691,A -85,B 0,C 180,E1 -304.845,E2 -304.845} C_VEL
LIN {X 0,Y 608.457,Z 273.693,A -85,B 0,C 180,E1 -307.747,E2 -307.747} C_VEL
LIN {X 0,Y 608.436,Z 273.696,A -85,B 0,C 180,E1 -310.327,E2 -310.327} C_VEL
LIN {X 0,Y 608.479,Z 273.691,A -85,B 0,C 180,E1 -313.309,E2 -313.309} C_VEL
LIN {X 0,Y 608.462,Z 273.695,A -85,B 0,C 180,E1 -316.13,E2 -316.13} C_VEL
LIN {X 0,Y 608.449,Z 273.698,A -85,B 0,C 180,E1 -318.823,E2 -318.823} C_VEL
LIN {X 0,Y 608.437,Z 273.699,A -85,B 0,C 180,E1 -321.409,E2 -321.409} C_VEL
LIN {X 0,Y 608.45,Z 273.697,A -85,B 0,C 180,E1 -323.955,E2 -323.955} C_VEL
LIN {X 0,Y 608.442,Z 273.853,A -85,B 0,C 180,E1 -325.312,E2 -325.312} C_VEL
LIN {X 0,Y 608.426,Z 278.888,A -85,B 0,C 180,E1 -327.903,E2 -327.903} C_VEL
LIN {X 0,Y 608.437,Z 283.344,A -85,B 0,C 180,E1 -330.219,E2 -330.219} C_VEL
LIN {X 0,Y 608.397,Z 288.889,A -85,B 0,C 180,E1 -333.223,E2 -333.223} C_VEL
LIN {X 0,Y 608.409,Z 293.036,A -85,B 0,C 180,E1 -335.427,E2 -335.427} C_VEL
LIN {X 0,Y 608.449,Z 298.565,A -85,B 0,C 180,E1 -338.308,E2 -338.308} C_VEL
LIN {X 0,Y 608.429,Z 304.425,A -85,B 0,C 180,E1 -341.297,E2 -341.297} C_VEL
LIN {X 0,Y 608.437,Z 309.624,A -85,B 0,C 180,E1 -343.905,E2 -343.905} C_VEL
LIN {X 0,Y 608.434,Z 315.154,A -85,B 0,C 180,E1 -346.643,E2 -346.643} C_VEL
LIN {X 0,Y 608.449,Z 318.524,A -85,B 0,C 180,E1 -348.296,E2 -348.296} C_VEL
LIN {X 0,Y 608.53,Z 334.397,A -85,B 0,C 180,E1 -348.677,E2 -348.677} C_VEL
LIN {X 0,Y 608.484,Z 346.476,A -85,B 0,C 180,E1 -349.099,E2 -349.099} C_VEL
LIN {X 0,Y 608.456,Z 358.936,A -85,B 0,C 180,E1 -349.686,E2 -349.686} C_VEL
LIN {X 0,Y 608.497,Z 370.067,A -85,B 0,C 180,E1 -350.359,E2 -350.359} C_VEL
LIN {X 0,Y 608.474,Z 379.084,A -85,B 0,C 180,E1 -351.029,E2 -351.029} C_VEL
LIN {X 0,Y 608.464,Z 388.349,A -85,B 0,C 180,E1 -351.866,E2 -351.866} C_VEL
LIN {X 0,Y 608.466,Z 397.323,A -85,B 0,C 180,E1 -352.867,E2 -352.867} C_VEL
LIN {X 0,Y 608.444,Z 404.556,A -85,B 0,C 180,E1 -353.866,E2 -353.866} C_VEL
LIN {X 0,Y 608.462,Z 409.435,A -85,B 0,C 180,E1 -354.698,E2 -354.698} C_VEL
LIN {X 0,Y 608.439,Z 414.179,A -85,B 0,C 180,E1 -355.694,E2 -355.694} C_VEL
LIN {X 0,Y 608.425,Z 417.812,A -85,B 0,C 180,E1 -356.689,E2 -356.689} C_VEL
LIN {X 0,Y 608.425,Z 419.69,A -85,B 0,C 180,E1 -357.352,E2 -357.352} C_VEL
LIN {X 0,Y 608.445,Z 421.126,A -85,B 0,C 180,E1 -358.014,E2 -358.014} C_VEL
LIN {X 0,Y 608.439,Z 422.752,A -85,B 0,C 180,E1 -359.338,E2 -359.338} C_VEL
LIN {X 0,Y 608.435,Z 422.995,A -85,B 0,C 180,E1 -360,E2 -360} C_VEL
LIN {X 0,Y 608.438,Z 422.815,A -85,B 0,C 180,E1 -360.662,E2 -360.662} C_VEL
LIN {X 0,Y 608.445,Z 421.275,A -85,B 0,C 180,E1 -361.986,E2 -361.986} C_VEL
LIN {X 0,Y 608.426,Z 419.919,A -85,B 0,C 180,E1 -362.648,E2 -362.648} C_VEL
LIN {X 0,Y 608.449,Z 417.042,A -85,B 0,C 180,E1 -363.642,E2 -363.642} C_VEL
LIN {X 0,Y 608.433,Z 413.143,A -85,B 0,C 180,E1 -364.638,E2 -364.638} C_VEL
LIN {X 0,Y 608.45,Z 408.112,A -85,B 0,C 180,E1 -365.634,E2 -365.634} C_VEL
LIN {X 0,Y 608.441,Z 401.791,A -85,B 0,C 180,E1 -366.633,E2 -366.633} C_VEL
LIN {X 0,Y 608.475,Z 393.88,A -85,B 0,C 180,E1 -367.633,E2 -367.633} C_VEL
LIN {X 0,Y 608.472,Z 384.036,A -85,B 0,C 180,E1 -368.636,E2 -368.636} C_VEL
LIN {X 0,Y 608.481,Z 373.707,A -85,B 0,C 180,E1 -369.473,E2 -369.473} C_VEL
LIN {X 0,Y 608.454,Z 362.095,A -85,B 0,C 180,E1 -370.229,E2 -370.229} C_VEL
LIN {X 0,Y 608.464,Z 350.47,A -85,B 0,C 180,E1 -370.821,E2 -370.821} C_VEL
LIN {X 0,Y 608.497,Z 338.309,A -85,B 0,C 180,E1 -371.289,E2 -371.289} C_VEL
LIN {X 0,Y 608.537,Z 325.547,A -85,B 0,C 180,E1 -371.639,E2 -371.639} C_VEL
LIN {X 0,Y 608.442,Z 318.536,A -85,B 0,C 180,E1 -371.789,E2 -371.789} C_VEL
LIN {X 0,Y 608.428,Z 313.954,A -85,B 0,C 180,E1 -374.038,E2 -374.038} C_VEL
LIN {X 0,Y 608.411,Z 308.422,A -85,B 0,C 180,E1 -376.785,E2 -376.785} C_VEL
LIN {X 0,Y 608.431,Z 302.89,A -85,B 0,C 180,E1 -379.571,E2 -379.571} C_VEL
LIN {X 0,Y 608.432,Z 297.237,A -85,B 0,C 180,E1 -382.469,E2 -382.469} C_VEL
LIN {X 0,Y 608.414,Z 293.207,A -85,B 0,C 180,E1 -384.573,E2 -384.573} C_VEL
LIN {X 0,Y 608.426,Z 288.272,A -85,B 0,C 180,E1 -387.197,E2 -387.197} C_VEL
LIN {X 0,Y 608.445,Z 283.049,A -85,B 0,C 180,E1 -389.967,E2 -389.967} C_VEL
LIN {X 0,Y 608.431,Z 277.314,A -85,B 0,C 180,E1 -392.517,E2 -392.517} C_VEL
LIN {X 0,Y 608.415,Z 273.701,A -85,B 0,C 180,E1 -393.972,E2 -393.972} C_VEL
LIN {X 0,Y 608.459,Z 273.693,A -85,B 0,C 180,E1 -396.915,E2 -396.915} C_VEL
LIN {X 0,Y 608.437,Z 273.696,A -85,B 0,C 180,E1 -399.442,E2 -399.442} C_VEL
LIN {X 0,Y 608.448,Z 273.695,A -85,B 0,C 180,E1 -402.063,E2 -402.063} C_VEL
LIN {X 0,Y 608.462,Z 273.693,A -85,B 0,C 180,E1 -404.795,E2 -404.795} C_VEL
LIN {X 0,Y 608.43,Z 273.696,A -85,B 0,C 180,E1 -407.669,E2 -407.669} C_VEL
LIN {X 0,Y 608.455,Z 273.697,A -85,B 0,C 180,E1 -409.697,E2 -409.697} C_VEL
LIN {X 0,Y 608.484,Z 273.69,A -85,B 0,C 180,E1 -412.84,E2 -412.84} C_VEL
LIN {X 0,Y 608.474,Z 273.825,A -85,B 0,C 180,E1 -414.273,E2 -414.273} C_VEL
LIN {X 0,Y 608.56,Z 281.668,A -85,B 0,C 180,E1 -416.335,E2 -416.335} C_VEL
LIN {X 0,Y 608.52,Z 292.467,A -85,B 0,C 180,E1 -419.087,E2 -419.087} C_VEL
LIN {X 0,Y 608.502,Z 303.154,A -85,B 0,C 180,E1 -421.736,E2 -421.736} C_VEL
LIN {X 0,Y 608.517,Z 313.627,A -85,B 0,C 180,E1 -424.271,E2 -424.271} C_VEL
LIN {X 0,Y 608.496,Z 326.177,A -85,B 0,C 180,E1 -427.237,E2 -427.237} C_VEL
LIN {X 0,Y 608.48,Z 338.453,A -85,B 0,C 180,E1 -430.079,E2 -430.079} C_VEL
LIN {X 0,Y 608.478,Z 350.731,A -85,B 0,C 180,E1 -432.871,E2 -432.871} C_VEL
LIN {X 0,Y 608.428,Z 363.009,A -85,B 0,C 180,E1 -435.62,E2 -435.62} C_VEL
LIN {X 0,Y 608.44,Z 374.712,A -85,B 0,C 180,E1 -438.211,E2 -438.211} C_VEL
LIN {X 0,Y 608.54,Z 388.179,A -85,B 0,C 180,E1 -438.466,E2 -438.466} C_VEL
LIN {X 0,Y 608.501,Z 400.488,A -85,B 0,C 180,E1 -438.827,E2 -438.827} C_VEL
LIN {X 0,Y 608.466,Z 411.856,A -85,B 0,C 180,E1 -439.287,E2 -439.287} C_VEL
LIN {X 0,Y 608.488,Z 422.754,A -85,B 0,C 180,E1 -439.855,E2 -439.855} C_VEL
LIN {X 0,Y 608.504,Z 434.251,A -85,B 0,C 180,E1 -440.611,E2 -440.611} C_VEL
LIN {X 0,Y 608.472,Z 443.535,A -85,B 0,C 180,E1 -441.364,E2 -441.364} C_VEL
LIN {X 0,Y 608.456,Z 451.989,A -85,B 0,C 180,E1 -442.2,E2 -442.2} C_VEL
LIN {X 0,Y 608.462,Z 460.235,A -85,B 0,C 180,E1 -443.201,E2 -443.201} C_VEL
LIN {X 0,Y 608.438,Z 466.876,A -85,B 0,C 180,E1 -444.199,E2 -444.199} C_VEL
LIN {X 0,Y 608.432,Z 472.95,A -85,B 0,C 180,E1 -445.362,E2 -445.362} C_VEL
LIN {X 0,Y 608.449,Z 476.896,A -85,B 0,C 180,E1 -446.358,E2 -446.358} C_VEL
LIN {X 0,Y 608.425,Z 479.809,A -85,B 0,C 180,E1 -447.352,E2 -447.352} C_VEL
LIN {X 0,Y 608.445,Z 481.201,A -85,B 0,C 180,E1 -448.014,E2 -448.014} C_VEL
LIN {X 0,Y 608.438,Z 482.783,A -85,B 0,C 180,E1 -449.338,E2 -449.338} C_VEL
LIN {X 0,Y 608.434,Z 483,A -85,B 0,C 180,E1 -450,E2 -450} C_VEL
LIN {X 0,Y 608.448,Z 482.184,A -85,B 0,C 180,E1 -451.324,E2 -451.324} C_VEL
LIN {X 0,Y 608.445,Z 481.201,A -85,B 0,C 180,E1 -451.986,E2 -451.986} C_VEL
LIN {X 0,Y 608.425,Z 479.809,A -85,B 0,C 180,E1 -452.648,E2 -452.648} C_VEL
LIN {X 0,Y 608.449,Z 476.896,A -85,B 0,C 180,E1 -453.642,E2 -453.642} C_VEL
LIN {X 0,Y 608.432,Z 472.95,A -85,B 0,C 180,E1 -454.638,E2 -454.638} C_VEL
LIN {X 0,Y 608.438,Z 466.876,A -85,B 0,C 180,E1 -455.801,E2 -455.801} C_VEL
LIN {X 0,Y 608.462,Z 460.235,A -85,B 0,C 180,E1 -456.799,E2 -456.799} C_VEL
LIN {X 0,Y 608.456,Z 451.989,A -85,B 0,C 180,E1 -457.8,E2 -457.8} C_VEL
LIN {X 0,Y 608.472,Z 443.536,A -85,B 0,C 180,E1 -458.636,E2 -458.636} C_VEL
LIN {X 0,Y 608.48,Z 433.09,A -85,B 0,C 180,E1 -459.473,E2 -459.473} C_VEL
LIN {X 0,Y 608.488,Z 422.754,A -85,B 0,C 180,E1 -460.145,E2 -460.145} C_VEL
LIN {X 0,Y 608.466,Z 411.856,A -85,B 0,C 180,E1 -460.713,E2 -460.713} C_VEL
LIN {X 0,Y 608.493,Z 400.086,A -85,B 0,C 180,E1 -461.186,E2 -461.186} C_VEL
LIN {X 0,Y 608.551,Z 387.264,A -85,B 0,C 180,E1 -461.554,E2 -461.554} C_VEL
LIN {X 0,Y 608.441,Z 374.712,A -85,B 0,C 180,E1 -461.789,E2 -461.789} C_VEL
LIN {X 0,Y 608.427,Z 363.009,A -85,B 0,C 180,E1 -464.38,E2 -464.38} C_VEL
LIN {X 0,Y 608.478,Z 350.731,A -85,B 0,C 180,E1 -467.129,E2 -467.129} C_VEL
LIN {X 0,Y 608.482,Z 338.453,A -85,B 0,C 180,E1 -469.921,E2 -469.921} C_VEL
LIN {X 0,Y 608.496,Z 326.177,A -85,B 0,C 180,E1 -472.763,E2 -472.763} C_VEL
LIN {X 0,Y 608.517,Z 313.627,A -85,B 0,C 180,E1 -475.729,E2 -475.729} C_VEL
LIN {X 0,Y 608.502,Z 303.154,A -85,B 0,C 180,E1 -478.264,E2 -478.264} C_VEL
LIN {X 0,Y 608.52,Z 292.467,A -85,B 0,C 180,E1 -480.913,E2 -480.913} C_VEL
LIN {X 0,Y 608.546,Z 281.362,A -85,B 0,C 180,E1 -483.745,E2 -483.745} C_VEL
LIN {X 0,Y 608.45,Z 273.828,A -85,B 0,C 180,E1 -485.728,E2 -485.728} C_VEL
LIN {X 0,Y 608.425,Z 273.693,A -85,B 0,C 180,E1 -488.235,E2 -488.235} C_VEL
LIN {X 0,Y 608.449,Z 273.693,A -85,B 0,C 180,E1 -491.177,E2 -491.177} C_VEL
LIN {X 0,Y 608.438,Z 273.691,A -85,B 0,C 180,E1 -493.873,E2 -493.873} C_VEL
LIN {X 0,Y 608.481,Z 273.691,A -85,B 0,C 180,E1 -496.69,E2 -496.69} C_VEL
LIN {X 0,Y 608.458,Z 273.69,A -85,B 0,C 180,E1 -498.824,E2 -498.824} C_VEL
LIN {X 0,Y 608.433,Z 273.691,A -85,B 0,C 180,E1 -501.409,E2 -501.409} C_VEL
LIN {X 0,Y 608.449,Z 273.697,A -85,B 0,C 180,E1 -503.955,E2 -503.955} C_VEL
LIN {X 0,Y 608.467,Z 273.69,A -85,B 0,C 180,E1 -506.329,E2 -506.329} C_VEL
LIN {X 0,Y 608.449,Z 273.689,A -85,B 0,C 180,E1 -508.733,E2 -508.733} C_VEL
LIN {X 0,Y 608.477,Z 273.691,A -85,B 0,C 180,E1 -511.38,E2 -511.38} C_VEL
LIN {X 0,Y 608.442,Z 273.692,A -85,B 0,C 180,E1 -513.964,E2 -513.964} C_VEL
LIN {X 0,Y 608.417,Z 273.702,A -85,B 0,C 180,E1 -515.427,E2 -515.427} C_VEL
LIN {X 0,Y 608.417,Z 276.294,A -85,B 0,C 180,E1 -517.592,E2 -517.592} C_VEL
LIN {X 0,Y 608.408,Z 279.81,A -85,B 0,C 180,E1 -520.428,E2 -520.428} C_VEL
LIN {X 0,Y 608.403,Z 283.325,A -85,B 0,C 180,E1 -523.215,E2 -523.215} C_VEL
LIN {X 0,Y 608.401,Z 286.904,A -85,B 0,C 180,E1 -526.01,E2 -526.01} C_VEL
LIN {X 0,Y 608.438,Z 289.949,A -85,B 0,C 180,E1 -528.338,E2 -528.338} C_VEL
LIN {X 0,Y 608.523,Z 303.623,A -85,B 0,C 180,E1 -528.656,E2 -528.656} C_VEL
LIN {X 0,Y 608.468,Z 315.15,A -85,B 0,C 180,E1 -529.046,E2 -529.046} C_VEL
LIN {X 0,Y 608.455,Z 327.369,A -85,B 0,C 180,E1 -529.602,E2 -529.602} C_VEL
LIN {X 0,Y 608.505,Z 338.788,A -85,B 0,C 180,E1 -530.275,E2 -530.275} C_VEL
LIN {X 0,Y 608.474,Z 349.081,A -85,B 0,C 180,E1 -531.029,E2 -531.029} C_VEL
LIN {X 0,Y 608.464,Z 358.351,A -85,B 0,C 180,E1 -531.866,E2 -531.866} C_VEL
LIN {X 0,Y 608.466,Z 367.325,A -85,B 0,C 180,E1 -532.867,E2 -532.867} C_VEL
LIN {X 0,Y 608.444,Z 374.556,A -85,B 0,C 180,E1 -533.867,E2 -533.867} C_VEL
LIN {X 0,Y 608.462,Z 379.434,A -85,B 0,C 180,E1 -534.698,E2 -534.698} C_VEL
LIN {X 0,Y 608.439,Z 384.178,A -85,B 0,C 180,E1 -535.694,E2 -535.694} C_VEL
LIN {X 0,Y 608.425,Z 387.811,A -85,B 0,C 180,E1 -536.689,E2 -536.689} C_VEL
LIN {X 0,Y 608.425,Z 389.691,A -85,B 0,C 180,E1 -537.352,E2 -537.352} C_VEL
LIN {X 0,Y 608.445,Z 391.127,A -85,B 0,C 180,E1 -538.014,E2 -538.014} C_VEL
LIN {X 0,Y 608.439,Z 392.752,A -85,B 0,C 180,E1 -539.338,E2 -539.338} C_VEL
LIN {X 0,Y 608.435,Z 392.995,A -85,B 0,C 180,E1 -540,E2 -540} C_VEL
LIN {X 0,Y 608.438,Z 392.815,A -85,B 0,C 180,E1 -540.662,E2 -540.662} C_VEL
LIN {X 0,Y 608.445,Z 391.276,A -85,B 0,C 180,E1 -541.986,E2 -541.986} C_VEL
LIN {X 0,Y 608.426,Z 389.917,A -85,B 0,C 180,E1 -542.648,E2 -542.648} C_VEL
LIN {X 0,Y 608.449,Z 387.04,A -85,B 0,C 180,E1 -543.642,E2 -543.642} C_VEL
LIN {X 0,Y 608.433,Z 383.142,A -85,B 0,C 180,E1 -544.638,E2 -544.638} C_VEL
LIN {X 0,Y 608.45,Z 378.112,A -85,B 0,C 180,E1 -545.634,E2 -545.634} C_VEL
LIN {X 0,Y 608.441,Z 371.794,A -85,B 0,C 180,E1 -546.633,E2 -546.633} C_VEL
LIN {X 0,Y 608.475,Z 363.875,A -85,B 0,C 180,E1 -547.633,E2 -547.633} C_VEL
LIN {X 0,Y 608.472,Z 354.031,A -85,B 0,C 180,E1 -548.636,E2 -548.636} C_VEL
LIN {X 0,Y 608.477,Z 351.937,A -85,B 0,C 180,E1 -548.819,E2 -548.819} C_VEL
LIN {X 0,Y 607.801,Z 347.593,A -85,B 0,C 180,E1 -549.19,E2 -549.19} C_VEL
LIN {X 0,Y 604.926,Z 340.343,A -85,B 0,C 180,E1 -549.769,E2 -549.769} C_VEL
LIN {X 0,Y 602.088,Z 332.706,A -85,B 0,C 180,E1 -550.302,E2 -550.302} C_VEL
LIN {X 0,Y 601.471,Z 327.65,A -85,B 0,C 180,E1 -550.595,E2 -550.595} C_VEL
LIN {X 0,Y 601.503,Z 315.573,A -85,B 0,C 180,E1 -551.157,E2 -551.157} C_VEL
LIN {X 0,Y 601.573,Z 303.02,A -85,B 0,C 180,E1 -551.584,E2 -551.584} C_VEL
LIN {X 0,Y 601.419,Z 290.795,A -85,B 0,C 180,E1 -551.875,E2 -551.875} C_VEL
LIN {X 0,Y 601.332,Z 289.869,A -85,B 0,C 180,E1 -551.93,E2 -551.93} C_VEL
LIN {X 0,Y 601.307,Z 286.956,A -85,B 0,C 180,E1 -554.208,E2 -554.208} C_VEL
LIN {X 0,Y 601.325,Z 283.439,A -85,B 0,C 180,E1 -556.989,E2 -556.989} C_VEL
LIN {X 0,Y 601.304,Z 279.922,A -85,B 0,C 180,E1 -559.813,E2 -559.813} C_VEL
LIN {X 0,Y 601.319,Z 276.53,A -85,B 0,C 180,E1 -562.583,E2 -562.583} C_VEL
LIN {X 0,Y 601.342,Z 274.581,A -85,B 0,C 180,E1 -564.272,E2 -564.272} C_VEL
LIN {X 0,Y 601.397,Z 274.572,A -85,B 0,C 180,E1 -566.364,E2 -566.364} C_VEL
LIN {X 0,Y 601.44,Z 274.568,A -85,B 0,C 180,E1 -568.789,E2 -568.789} C_VEL
LIN {X 0,Y 601.404,Z 274.567,A -85,B 0,C 180,E1 -571.727,E2 -571.727} C_VEL
LIN {X 0,Y 601.421,Z 274.57,A -85,B 0,C 180,E1 -574.119,E2 -574.119} C_VEL
LIN {X 0,Y 601.404,Z 274.571,A -85,B 0,C 180,E1 -576.583,E2 -576.583} C_VEL
LIN {X 0,Y 601.418,Z 274.564,A -85,B 0,C 180,E1 -579.126,E2 -579.126} C_VEL
LIN {X 0,Y 601.428,Z 274.569,A -85,B 0,C 180,E1 -581.765,E2 -581.765} C_VEL
LIN {X 0,Y 601.429,Z 274.565,A -85,B 0,C 180,E1 -584.535,E2 -584.535} C_VEL
LIN {X 0,Y 601.416,Z 274.568,A -85,B 0,C 180,E1 -587.409,E2 -587.409} C_VEL
LIN {X 0,Y 601.404,Z 274.571,A -85,B 0,C 180,E1 -590.004,E2 -590.004} C_VEL
LIN {X 0,Y 601.439,Z 274.562,A -85,B 0,C 180,E1 -592.618,E2 -592.618} C_VEL
LIN {X 0,Y 601.399,Z 274.658,A -85,B 0,C 180,E1 -595.474,E2 -595.474} C_VEL
LIN {X 0,Y 601.373,Z 280.704,A -85,B 0,C 180,E1 -598.553,E2 -598.553} C_VEL
LIN {X 0,Y 601.317,Z 286.069,A -85,B 0,C 180,E1 -601.367,E2 -601.367} C_VEL
LIN {X 0,Y 601.34,Z 290.273,A -85,B 0,C 180,E1 -603.633,E2 -603.633} C_VEL
LIN {X 0,Y 601.366,Z 295.802,A -85,B 0,C 180,E1 -606.587,E2 -606.587} C_VEL
LIN {X 0,Y 601.344,Z 301.331,A -85,B 0,C 180,E1 -609.475,E2 -609.475} C_VEL
LIN {X 0,Y 601.338,Z 306.861,A -85,B 0,C 180,E1 -612.31,E2 -612.31} C_VEL
LIN {X 0,Y 601.335,Z 312.391,A -85,B 0,C 180,E1 -615.101,E2 -615.101} C_VEL
LIN {X 0,Y 601.349,Z 318.266,A -85,B 0,C 180,E1 -618.027,E2 -618.027} C_VEL
LIN {X 0,Y 601.341,Z 318.757,A -85,B 0,C 180,E1 -618.177,E2 -618.177} C_VEL
LIN {X 0,Y 601.593,Z 325.323,A -85,B 0,C 180,E1 -618.31,E2 -618.31} C_VEL
LIN {X 0,Y 601.555,Z 338.16,A -85,B 0,C 180,E1 -618.665,E2 -618.665} C_VEL
LIN {X 0,Y 601.486,Z 350.163,A -85,B 0,C 180,E1 -619.13,E2 -619.13} C_VEL
LIN {X 0,Y 601.481,Z 362.008,A -85,B 0,C 180,E1 -619.736,E2 -619.736} C_VEL
LIN {X 0,Y 601.462,Z 373.63,A -85,B 0,C 180,E1 -620.5,E2 -620.5} C_VEL
LIN {X 0,Y 601.436,Z 383.011,A -85,B 0,C 180,E1 -621.262,E2 -621.262} C_VEL
LIN {X 0,Y 601.4,Z 391.587,A -85,B 0,C 180,E1 -622.108,E2 -622.108} C_VEL
LIN {X 0,Y 601.388,Z 399.908,A -85,B 0,C 180,E1 -623.12,E2 -623.12} C_VEL
LIN {X 0,Y 601.373,Z 406.608,A -85,B 0,C 180,E1 -624.131,E2 -624.131} C_VEL
LIN {X 0,Y 601.335,Z 412.744,A -85,B 0,C 180,E1 -625.307,E2 -625.307} C_VEL
LIN {X 0,Y 601.367,Z 416.735,A -85,B 0,C 180,E1 -626.315,E2 -626.315} C_VEL
LIN {X 0,Y 601.324,Z 419.686,A -85,B 0,C 180,E1 -627.32,E2 -627.32} C_VEL
LIN {X 0,Y 601.343,Z 421.121,A -85,B 0,C 180,E1 -627.991,E2 -627.991} C_VEL
LIN {X 0,Y 601.347,Z 422.133,A -85,B 0,C 180,E1 -628.661,E2 -628.661} C_VEL
LIN {X 0,Y 601.336,Z 422.991,A -85,B 0,C 180,E1 -630,E2 -630} C_VEL
LIN {X 0,Y 601.339,Z 422.814,A -85,B 0,C 180,E1 -630.67,E2 -630.67} C_VEL
LIN {X 0,Y 601.344,Z 421.273,A -85,B 0,C 180,E1 -632.009,E2 -632.009} C_VEL
LIN {X 0,Y 601.326,Z 419.917,A -85,B 0,C 180,E1 -632.68,E2 -632.68} C_VEL
LIN {X 0,Y 601.368,Z 417.043,A -85,B 0,C 180,E1 -633.685,E2 -633.685} C_VEL
LIN {X 0,Y 601.337,Z 413.143,A -85,B 0,C 180,E1 -634.693,E2 -634.693} C_VEL
LIN {X 0,Y 601.373,Z 408.109,A -85,B 0,C 180,E1 -635.701,E2 -635.701} C_VEL
LIN {X 0,Y 601.382,Z 401.779,A -85,B 0,C 180,E1 -636.711,E2 -636.711} C_VEL
LIN {X 0,Y 601.396,Z 393.878,A -85,B 0,C 180,E1 -637.723,E2 -637.723} C_VEL
LIN {X 0,Y 601.437,Z 384.025,A -85,B 0,C 180,E1 -638.738,E2 -638.738} C_VEL
LIN {X 0,Y 601.449,Z 373.701,A -85,B 0,C 180,E1 -639.585,E2 -639.585} C_VEL
LIN {X 0,Y 601.452,Z 362.09,A -85,B 0,C 180,E1 -640.35,E2 -640.35} C_VEL
LIN {X 0,Y 601.488,Z 349.932,A -85,B 0,C 180,E1 -640.97,E2 -640.97} C_VEL
LIN {X 0,Y 601.549,Z 337.214,A -85,B 0,C 180,E1 -641.456,E2 -641.456} C_VEL
LIN {X 0,Y 601.61,Z 324.603,A -85,B 0,C 180,E1 -641.796,E2 -641.796} C_VEL
LIN {X 0,Y 601.339,Z 318.534,A -85,B 0,C 180,E1 -641.93,E2 -641.93} C_VEL
LIN {X 0,Y 601.332,Z 312.57,A -85,B 0,C 180,E1 -644.899,E2 -644.899} C_VEL
LIN {X 0,Y 601.332,Z 307.038,A -85,B 0,C 180,E1 -647.69,E2 -647.69} C_VEL
LIN {X 0,Y 601.346,Z 301.505,A -85,B 0,C 180,E1 -650.525,E2 -650.525} C_VEL
LIN {X 0,Y 601.366,Z 295.972,A -85,B 0,C 180,E1 -653.413,E2 -653.413} C_VEL
LIN {X 0,Y 601.343,Z 290.439,A -85,B 0,C 180,E1 -656.367,E2 -656.367} C_VEL
LIN {X 0,Y 601.327,Z 285.982,A -85,B 0,C 180,E1 -658.769,E2 -658.769} C_VEL
LIN {X 0,Y 601.373,Z 280.884,A -85,B 0,C 180,E1 -661.447,E2 -661.447} C_VEL
LIN {X 0,Y 601.366,Z 275.661,A -85,B 0,C 180,E1 -664.123,E2 -664.123} C_VEL
LIN {X 0,Y 601.4,Z 274.575,A -85,B 0,C 180,E1 -664.729,E2 -664.729} C_VEL
LIN {X 0,Y 601.435,Z 274.57,A -85,B 0,C 180,E1 -667.419,E2 -667.419} C_VEL
LIN {X 0,Y 601.416,Z 274.572,A -85,B 0,C 180,E1 -669.995,E2 -669.995} C_VEL
LIN {X 0,Y 601.417,Z 274.572,A -85,B 0,C 180,E1 -672.67,E2 -672.67} C_VEL
LIN {X 0,Y 601.402,Z 274.572,A -85,B 0,C 180,E1 -675.479,E2 -675.479} C_VEL
LIN {X 0,Y 601.418,Z 274.57,A -85,B 0,C 180,E1 -678.408,E2 -678.408} C_VEL
LIN {X 0,Y 601.435,Z 274.568,A -85,B 0,C 180,E1 -680.875,E2 -680.875} C_VEL
LIN {X 0,Y 601.399,Z 274.572,A -85,B 0,C 180,E1 -683.417,E2 -683.417} C_VEL
LIN {X 0,Y 601.397,Z 274.627,A -85,B 0,C 180,E1 -685.372,E2 -685.372} C_VEL
LIN {X 0,Y 601.373,Z 280.774,A -85,B 0,C 180,E1 -688.553,E2 -688.553} C_VEL
LIN {X 0,Y 601.319,Z 286.108,A -85,B 0,C 180,E1 -691.367,E2 -691.367} C_VEL
LIN {X 0,Y 601.34,Z 290.273,A -85,B 0,C 180,E1 -693.633,E2 -693.633} C_VEL
LIN {X 0,Y 601.366,Z 295.802,A -85,B 0,C 180,E1 -696.587,E2 -696.587} C_VEL
LIN {X 0,Y 601.344,Z 301.331,A -85,B 0,C 180,E1 -699.475,E2 -699.475} C_VEL
LIN {X 0,Y 601.338,Z 306.861,A -85,B 0,C 180,E1 -702.31,E2 -702.31} C_VEL
LIN {X 0,Y 601.335,Z 312.39,A -85,B 0,C 180,E1 -705.101,E2 -705.101} C_VEL
LIN {X 0,Y 601.349,Z 318.266,A -85,B 0,C 180,E1 -708.027,E2 -708.027} C_VEL
LIN {X 0,Y 601.341,Z 318.782,A -85,B 0,C 180,E1 -708.177,E2 -708.177} C_VEL
LIN {X 0,Y 601.593,Z 325.305,A -85,B 0,C 180,E1 -708.31,E2 -708.31} C_VEL
LIN {X 0,Y 601.562,Z 337.856,A -85,B 0,C 180,E1 -708.655,E2 -708.655} C_VEL
LIN {X 0,Y 601.485,Z 350.189,A -85,B 0,C 180,E1 -709.13,E2 -709.13} C_VEL
LIN {X 0,Y 601.481,Z 361.986,A -85,B 0,C 180,E1 -709.736,E2 -709.736} C_VEL
LIN {X 0,Y 601.451,Z 372.466,A -85,B 0,C 180,E1 -710.415,E2 -710.415} C_VEL
LIN {X 0,Y 601.436,Z 383.017,A -85,B 0,C 180,E1 -711.262,E2 -711.262} C_VEL
LIN {X 0,Y 601.4,Z 391.59,A -85,B 0,C 180,E1 -712.108,E2 -712.108} C_VEL
LIN {X 0,Y 601.388,Z 399.904,A -85,B 0,C 180,E1 -713.12,E2 -713.12} C_VEL
LIN {X 0,Y 601.373,Z 406.603,A -85,B 0,C 180,E1 -714.131,E2 -714.131} C_VEL
LIN {X 0,Y 601.335,Z 412.749,A -85,B 0,C 180,E1 -715.307,E2 -715.307} C_VEL
LIN {X 0,Y 601.367,Z 416.739,A -85,B 0,C 180,E1 -716.315,E2 -716.315} C_VEL
LIN {X 0,Y 601.324,Z 419.69,A -85,B 0,C 180,E1 -717.32,E2 -717.32} C_VEL
LIN {X 0,Y 601.343,Z 421.124,A -85,B 0,C 180,E1 -717.991,E2 -717.991} C_VEL
LIN {X 0,Y 601.339,Z 422.753,A -85,B 0,C 180,E1 -719.33,E2 -719.33} C_VEL
LIN {X 0,Y 601.336,Z 422.988,A -85,B 0,C 180,E1 -720,E2 -720} C_VEL
LIN {X 0,Y 601.339,Z 422.813,A -85,B 0,C 180,E1 -720.67,E2 -720.67} C_VEL
LIN {X 0,Y 601.348,Z 422.238,A -85,B 0,C 180,E1 -721.339,E2 -721.339} C_VEL
LIN {X 0,Y 601.326,Z 419.916,A -85,B 0,C 180,E1 -722.68,E2 -722.68} C_VEL
LIN {X 0,Y 601.368,Z 417.043,A -85,B 0,C 180,E1 -723.685,E2 -723.685} C_VEL
LIN {X 0,Y 601.337,Z 413.143,A -85,B 0,C 180,E1 -724.693,E2 -724.693} C_VEL
LIN {X 0,Y 601.373,Z 408.11,A -85,B 0,C 180,E1 -725.701,E2 -725.701} C_VEL
LIN {X 0,Y 601.382,Z 401.778,A -85,B 0,C 180,E1 -726.711,E2 -726.711} C_VEL
LIN {X 0,Y 601.396,Z 393.878,A -85,B 0,C 180,E1 -727.723,E2 -727.723} C_VEL
LIN {X 0,Y 601.436,Z 384.03,A -85,B 0,C 180,E1 -728.738,E2 -728.738} C_VEL
LIN {X 0,Y 601.449,Z 373.691,A -85,B 0,C 180,E1 -729.585,E2 -729.585} C_VEL
LIN {X 0,Y 601.469,Z 363.493,A -85,B 0,C 180,E1 -730.264,E2 -730.264} C_VEL
LIN {X 0,Y 601.481,Z 352.192,A -85,B 0,C 180,E1 -730.868,E2 -730.868} C_VEL
LIN {X 0,Y 601.525,Z 339.69,A -85,B 0,C 180,E1 -731.375,E2 -731.375} C_VEL
LIN {X 0,Y 601.575,Z 326.424,A -85,B 0,C 180,E1 -731.754,E2 -731.754} C_VEL
LIN {X 0,Y 601.364,Z 319.052,A -85,B 0,C 180,E1 -731.908,E2 -731.908} C_VEL
LIN {X 0,Y 601.339,Z 318.535,A -85,B 0,C 180,E1 -731.93,E2 -731.93} C_VEL
LIN {X 0,Y 601.332,Z 312.57,A -85,B 0,C 180,E1 -734.899,E2 -734.899} C_VEL
LIN {X 0,Y 601.332,Z 307.038,A -85,B 0,C 180,E1 -737.69,E2 -737.69} C_VEL
LIN {X 0,Y 601.346,Z 301.505,A -85,B 0,C 180,E1 -740.525,E2 -740.525} C_VEL
LIN {X 0,Y 601.366,Z 295.973,A -85,B 0,C 180,E1 -743.413,E2 -743.413} C_VEL
LIN {X 0,Y 601.343,Z 290.439,A -85,B 0,C 180,E1 -746.367,E2 -746.367} C_VEL
LIN {X 0,Y 601.321,Z 285.906,A -85,B 0,C 180,E1 -748.768,E2 -748.768} C_VEL
LIN {X 0,Y 601.326,Z 281.292,A -85,B 0,C 180,E1 -750.947,E2 -750.947} C_VEL
LIN {X 0,Y 601.368,Z 274.88,A -85,B 0,C 180,E1 -753.621,E2 -753.621} C_VEL
LIN {X 0,Y 601.363,Z 274.58,A -85,B 0,C 180,E1 -753.925,E2 -753.925} C_VEL
LIN {X 0,Y 601.405,Z 274.575,A -85,B 0,C 180,E1 -756.583,E2 -756.583} C_VEL
LIN {X 0,Y 601.41,Z 274.571,A -85,B 0,C 180,E1 -759.532,E2 -759.532} C_VEL
LIN {X 0,Y 601.419,Z 274.574,A -85,B 0,C 180,E1 -761.766,E2 -761.766} C_VEL
LIN {X 0,Y 601.428,Z 274.571,A -85,B 0,C 180,E1 -764.535,E2 -764.535} C_VEL
LIN {X 0,Y 601.385,Z 274.575,A -85,B 0,C 180,E1 -767.327,E2 -767.327} C_VEL
LIN {X 0,Y 601.402,Z 274.573,A -85,B 0,C 180,E1 -770.004,E2 -770.004} C_VEL
LIN {X 0,Y 601.44,Z 274.568,A -85,B 0,C 180,E1 -772.618,E2 -772.618} C_VEL
LIN {X 0,Y 601.431,Z 274.697,A -85,B 0,C 180,E1 -774.024,E2 -774.024} C_VEL
LIN {X 0,Y 601.648,Z 278.598,A -85,B 0,C 180,E1 -775.083,E2 -775.083} C_VEL
LIN {X 0,Y 601.585,Z 287.807,A -85,B 0,C 180,E1 -777.493,E2 -777.493} C_VEL
LIN {X 0,Y 601.561,Z 297.015,A -85,B 0,C 180,E1 -779.843,E2 -779.843} C_VEL
LIN {X 0,Y 601.55,Z 308.151,A -85,B 0,C 180,E1 -782.613,E2 -782.613} C_VEL
LIN {X 0,Y 601.489,Z 318.502,A -85,B 0,C 180,E1 -785.125,E2 -785.125} C_VEL
LIN {X 0,Y 601.473,Z 329.362,A -85,B 0,C 180,E1 -787.709,E2 -787.709} C_VEL
LIN {X 0,Y 601.436,Z 341.523,A -85,B 0,C 180,E1 -790.547,E2 -790.547} C_VEL
LIN {X 0,Y 601.418,Z 353.882,A -85,B 0,C 180,E1 -793.382,E2 -793.382} C_VEL
LIN {X 0,Y 601.389,Z 366.371,A -85,B 0,C 180,E1 -796.204,E2 -796.204} C_VEL
LIN {X 0,Y 601.377,Z 374.712,A -85,B 0,C 180,E1 -798.071,E2 -798.071} C_VEL
LIN {X 0,Y 601.624,Z 386.351,A -85,B 0,C 180,E1 -798.289,E2 -798.289} C_VEL
LIN {X 0,Y 601.562,Z 399.234,A -85,B 0,C 180,E1 -798.655,E2 -798.655} C_VEL
LIN {X 0,Y 601.482,Z 411.24,A -85,B 0,C 180,E1 -799.132,E2 -799.132} C_VEL
LIN {X 0,Y 601.478,Z 422.755,A -85,B 0,C 180,E1 -799.736,E2 -799.736} C_VEL
LIN {X 0,Y 601.462,Z 434.251,A -85,B 0,C 180,E1 -800.5,E2 -800.5} C_VEL
LIN {X 0,Y 601.436,Z 443.536,A -85,B 0,C 180,E1 -801.262,E2 -801.262} C_VEL
LIN {X 0,Y 601.4,Z 451.989,A -85,B 0,C 180,E1 -802.108,E2 -802.108} C_VEL
LIN {X 0,Y 601.382,Z 460.235,A -85,B 0,C 180,E1 -803.12,E2 -803.12} C_VEL
LIN {X 0,Y 601.373,Z 466.877,A -85,B 0,C 180,E1 -804.131,E2 -804.131} C_VEL
LIN {X 0,Y 601.336,Z 472.95,A -85,B 0,C 180,E1 -805.307,E2 -805.307} C_VEL
LIN {X 0,Y 601.368,Z 476.896,A -85,B 0,C 180,E1 -806.315,E2 -806.315} C_VEL
LIN {X 0,Y 601.325,Z 479.809,A -85,B 0,C 180,E1 -807.32,E2 -807.32} C_VEL
LIN {X 0,Y 601.343,Z 481.201,A -85,B 0,C 180,E1 -807.991,E2 -807.991} C_VEL
LIN {X 0,Y 601.339,Z 482.784,A -85,B 0,C 180,E1 -809.33,E2 -809.33} C_VEL
LIN {X 0,Y 601.335,Z 483,A -85,B 0,C 180,E1 -810,E2 -810} C_VEL
LIN {X 0,Y 601.347,Z 482.184,A -85,B 0,C 180,E1 -811.339,E2 -811.339} C_VEL
LIN {X 0,Y 601.343,Z 481.202,A -85,B 0,C 180,E1 -812.009,E2 -812.009} C_VEL
LIN {X 0,Y 601.325,Z 479.809,A -85,B 0,C 180,E1 -812.68,E2 -812.68} C_VEL
LIN {X 0,Y 601.368,Z 476.896,A -85,B 0,C 180,E1 -813.685,E2 -813.685} C_VEL
LIN {X 0,Y 601.336,Z 472.95,A -85,B 0,C 180,E1 -814.693,E2 -814.693} C_VEL
LIN {X 0,Y 601.373,Z 466.877,A -85,B 0,C 180,E1 -815.869,E2 -815.869} C_VEL
LIN {X 0,Y 601.382,Z 460.235,A -85,B 0,C 180,E1 -816.88,E2 -816.88} C_VEL
LIN {X 0,Y 601.4,Z 451.989,A -85,B 0,C 180,E1 -817.892,E2 -817.892} C_VEL
LIN {X 0,Y 601.436,Z 443.536,A -85,B 0,C 180,E1 -818.738,E2 -818.738} C_VEL
LIN {X 0,Y 601.449,Z 433.09,A -85,B 0,C 180,E1 -819.585,E2 -819.585} C_VEL
LIN {X 0,Y 601.478,Z 422.755,A -85,B 0,C 180,E1 -820.264,E2 -820.264} C_VEL
LIN {X 0,Y 601.482,Z 411.232,A -85,B 0,C 180,E1 -820.869,E2 -820.869} C_VEL
LIN {X 0,Y 601.527,Z 398.334,A -85,B 0,C 180,E1 -821.375,E2 -821.375} C_VEL
LIN {X 0,Y 601.598,Z 385.436,A -85,B 0,C 180,E1 -821.733,E2 -821.733} C_VEL
LIN {X 0,Y 601.379,Z 374.712,A -85,B 0,C 180,E1 -821.929,E2 -821.929} C_VEL
LIN {X 0,Y 601.379,Z 363.009,A -85,B 0,C 180,E1 -824.552,E2 -824.552} C_VEL
LIN {X 0,Y 601.44,Z 350.731,A -85,B 0,C 180,E1 -827.336,E2 -827.336} C_VEL
LIN {X 0,Y 601.467,Z 338.453,A -85,B 0,C 180,E1 -830.164,E2 -830.164} C_VEL
LIN {X 0,Y 601.497,Z 326.175,A -85,B 0,C 180,E1 -833.043,E2 -833.043} C_VEL
LIN {X 0,Y 601.531,Z 314.289,A -85,B 0,C 180,E1 -835.89,E2 -835.89} C_VEL
LIN {X 0,Y 601.538,Z 303.154,A -85,B 0,C 180,E1 -838.621,E2 -838.621} C_VEL
LIN {X 0,Y 601.629,Z 291.763,A -85,B 0,C 180,E1 -841.487,E2 -841.487} C_VEL
LIN {X 0,Y 601.613,Z 281.668,A -85,B 0,C 180,E1 -844.107,E2 -844.107} C_VEL
LIN {X 0,Y 601.571,Z 275.529,A -85,B 0,C 180,E1 -845.742,E2 -845.742} C_VEL
LIN {X 0,Y 601.381,Z 274.575,A -85,B 0,C 180,E1 -846.021,E2 -846.021} C_VEL
LIN {X 0,Y 601.393,Z 274.571,A -85,B 0,C 180,E1 -848.466,E2 -848.466} C_VEL
LIN {X 0,Y 601.409,Z 274.575,A -85,B 0,C 180,E1 -850.875,E2 -850.875} C_VEL
LIN {X 0,Y 601.406,Z 274.567,A -85,B 0,C 180,E1 -853.589,E2 -853.589} C_VEL
LIN {X 0,Y 601.431,Z 274.572,A -85,B 0,C 180,E1 -856.427,E2 -856.427} C_VEL
LIN {X 0,Y 601.407,Z 274.566,A -85,B 0,C 180,E1 -859.428,E2 -859.428} C_VEL
LIN {X 0,Y 601.411,Z 274.569,A -85,B 0,C 180,E1 -861.731,E2 -861.731} C_VEL
LIN {X 0,Y 601.388,Z 274.575,A -85,B 0,C 180,E1 -864.245,E2 -864.245} C_VEL
LIN {X 0,Y 601.429,Z 274.564,A -85,B 0,C 180,E1 -866.686,E2 -866.686} C_VEL
LIN {X 0,Y 601.415,Z 274.566,A -85,B 0,C 180,E1 -869.058,E2 -869.058} C_VEL
LIN {X 0,Y 601.436,Z 274.569,A -85,B 0,C 180,E1 -871.373,E2 -871.373} C_VEL
LIN {X 0,Y 601.401,Z 274.574,A -85,B 0,C 180,E1 -873.636,E2 -873.636} C_VEL
LIN {X 0,Y 601.334,Z 274.582,A -85,B 0,C 180,E1 -875.854,E2 -875.854} C_VEL
LIN {X 0,Y 601.328,Z 277.174,A -85,B 0,C 180,E1 -878.037,E2 -878.037} C_VEL
LIN {X 0,Y 601.306,Z 279.81,A -85,B 0,C 180,E1 -880.187,E2 -880.187} C_VEL
LIN {X 0,Y 601.327,Z 283.326,A -85,B 0,C 180,E1 -883.011,E2 -883.011} C_VEL
LIN {X 0,Y 601.327,Z 287.037,A -85,B 0,C 180,E1 -885.946,E2 -885.946} C_VEL
LIN {X 0,Y 601.338,Z 289.991,A -85,B 0,C 180,E1 -888.198,E2 -888.198} C_VEL
LIN {X 0,Y 601.592,Z 297.186,A -85,B 0,C 180,E1 -888.353,E2 -888.353} C_VEL
LIN {X 0,Y 601.543,Z 310.611,A -85,B 0,C 180,E1 -888.747,E2 -888.747} C_VEL
LIN {X 0,Y 601.48,Z 322.234,A -85,B 0,C 180,E1 -889.225,E2 -889.225} C_VEL
LIN {X 0,Y 601.467,Z 333.42,A -85,B 0,C 180,E1 -889.821,E2 -889.821} C_VEL
LIN {X 0,Y 601.456,Z 344.8,A -85,B 0,C 180,E1 -890.585,E2 -890.585} C_VEL
LIN {X 0,Y 601.424,Z 354.854,A -85,B 0,C 180,E1 -891.432,E2 -891.432} C_VEL
LIN {X 0,Y 601.396,Z 363.07,A -85,B 0,C 180,E1 -892.277,E2 -892.277} C_VEL
LIN {X 0,Y 601.383,Z 371.136,A -85,B 0,C 180,E1 -893.289,E2 -893.289} C_VEL
LIN {X 0,Y 601.372,Z 377.612,A -85,B 0,C 180,E1 -894.299,E2 -894.299} C_VEL
LIN {X 0,Y 601.335,Z 382.753,A -85,B 0,C 180,E1 -895.307,E2 -895.307} C_VEL
LIN {X 0,Y 601.367,Z 386.743,A -85,B 0,C 180,E1 -896.315,E2 -896.315} C_VEL
LIN {X 0,Y 601.324,Z 389.695,A -85,B 0,C 180,E1 -897.32,E2 -897.32} C_VEL
LIN {X 0,Y 601.344,Z 391.13,A -85,B 0,C 180,E1 -897.991,E2 -897.991} C_VEL
LIN {X 0,Y 601.339,Z 392.753,A -85,B 0,C 180,E1 -899.33,E2 -899.33} C_VEL
LIN {X 0,Y 601.336,Z 392.996,A -85,B 0,C 180,E1 -900,E2 -900} C_VEL
LIN {X 0,Y 601.339,Z 392.816,A -85,B 0,C 180,E1 -900.67,E2 -900.67} C_VEL
LIN {X 0,Y 601.344,Z 391.277,A -85,B 0,C 180,E1 -902.009,E2 -902.009} C_VEL
LIN {X 0,Y 601.326,Z 389.909,A -85,B 0,C 180,E1 -902.68,E2 -902.68} C_VEL
LIN {X 0,Y 601.368,Z 387.033,A -85,B 0,C 180,E1 -903.685,E2 -903.685} C_VEL
LIN {X 0,Y 601.337,Z 383.137,A -85,B 0,C 180,E1 -904.693,E2 -904.693} C_VEL
LIN {X 0,Y 601.373,Z 378.109,A -85,B 0,C 180,E1 -905.701,E2 -905.701} C_VEL
LIN {X 0,Y 601.382,Z 371.79,A -85,B 0,C 180,E1 -906.711,E2 -906.711} C_VEL
LIN {X 0,Y 601.396,Z 363.865,A -85,B 0,C 180,E1 -907.723,E2 -907.723} C_VEL
LIN {X 0,Y 601.421,Z 355.795,A -85,B 0,C 180,E1 -908.569,E2 -908.569} C_VEL
LIN {X 0,Y 601.453,Z 345.963,A -85,B 0,C 180,E1 -909.415,E2 -909.415} C_VEL
LIN {X 0,Y 601.463,Z 334.917,A -85,B 0,C 180,E1 -910.18,E2 -910.18} C_VEL
LIN {X 0,Y 601.471,Z 327.65,A -85,B 0,C 180,E1 -910.595,E2 -910.595} C_VEL
LIN {X 0,Y 600.871,Z 322.517,A -85,B 0,C 180,E1 -910.867,E2 -910.867} C_VEL
LIN {X 0,Y 598.105,Z 314.043,A -85,B 0,C 180,E1 -911.281,E2 -911.281} C_VEL
LIN {X 0,Y 595.346,Z 305.29,A -85,B 0,C 180,E1 -911.641,E2 -911.641} C_VEL
LIN {X 0,Y 594.63,Z 299.721,A -85,B 0,C 180,E1 -911.813,E2 -911.813} C_VEL
LIN {X 0,Y 594.521,Z 291.776,A -85,B 0,C 180,E1 -911.996,E2 -911.996} C_VEL
LIN {X 0,Y 594.229,Z 289.896,A -85,B 0,C 180,E1 -912.053,E2 -912.053} C_VEL
LIN {X 0,Y 594.201,Z 286.956,A -85,B 0,C 180,E1 -914.382,E2 -914.382} C_VEL
LIN {X 0,Y 594.229,Z 283.438,A -85,B 0,C 180,E1 -917.198,E2 -917.198} C_VEL
LIN {X 0,Y 594.209,Z 279.921,A -85,B 0,C 180,E1 -920.06,E2 -920.06} C_VEL
LIN {X 0,Y 594.233,Z 276.725,A -85,B 0,C 180,E1 -922.704,E2 -922.704} C_VEL
LIN {X 0,Y 594.229,Z 275.524,A -85,B 0,C 180,E1 -923.711,E2 -923.711} C_VEL
LIN {X 0,Y 594.381,Z 275.442,A -85,B 0,C 180,E1 -926.021,E2 -926.021} C_VEL
LIN {X 0,Y 594.384,Z 275.444,A -85,B 0,C 180,E1 -928.999,E2 -928.999} C_VEL
LIN {X 0,Y 594.38,Z 275.441,A -85,B 0,C 180,E1 -931.643,E2 -931.643} C_VEL
LIN {X 0,Y 594.378,Z 275.447,A -85,B 0,C 180,E1 -934.58,E2 -934.58} C_VEL
LIN {X 0,Y 594.394,Z 275.441,A -85,B 0,C 180,E1 -937.609,E2 -937.609} C_VEL
LIN {X 0,Y 594.373,Z 275.445,A -85,B 0,C 180,E1 -940.567,E2 -940.567} C_VEL
LIN {X 0,Y 594.37,Z 275.444,A -85,B 0,C 180,E1 -943.3,E2 -943.3} C_VEL
LIN {X 0,Y 594.372,Z 275.447,A -85,B 0,C 180,E1 -946.16,E2 -946.16} C_VEL
LIN {X 0,Y 594.382,Z 275.441,A -85,B 0,C 180,E1 -948.536,E2 -948.536} C_VEL
LIN {X 0,Y 594.385,Z 275.445,A -85,B 0,C 180,E1 -951.296,E2 -951.296} C_VEL
LIN {X 0,Y 594.352,Z 275.452,A -85,B 0,C 180,E1 -953.755,E2 -953.755} C_VEL
LIN {X 0,Y 594.346,Z 275.526,A -85,B 0,C 180,E1 -955.546,E2 -955.546} C_VEL
LIN {X 0,Y 594.322,Z 281.54,A -85,B 0,C 180,E1 -958.647,E2 -958.647} C_VEL
LIN {X 0,Y 594.271,Z 287.426,A -85,B 0,C 180,E1 -961.767,E2 -961.767} C_VEL
LIN {X 0,Y 594.292,Z 293.039,A -85,B 0,C 180,E1 -964.803,E2 -964.803} C_VEL
LIN {X 0,Y 594.276,Z 298.568,A -85,B 0,C 180,E1 -967.763,E2 -967.763} C_VEL
LIN {X 0,Y 594.244,Z 302.715,A -85,B 0,C 180,E1 -969.942,E2 -969.942} C_VEL
LIN {X 0,Y 594.245,Z 306.862,A -85,B 0,C 180,E1 -972.092,E2 -972.092} C_VEL
LIN {X 0,Y 594.252,Z 311.009,A -85,B 0,C 180,E1 -974.216,E2 -974.216} C_VEL
LIN {X 0,Y 594.227,Z 316.539,A -85,B 0,C 180,E1 -977.014,E2 -977.014} C_VEL
LIN {X 0,Y 594.262,Z 318.738,A -85,B 0,C 180,E1 -978.034,E2 -978.034} C_VEL
LIN {X 0,Y 594.66,Z 323.435,A -85,B 0,C 180,E1 -978.129,E2 -978.129} C_VEL
LIN {X 0,Y 594.592,Z 335.789,A -85,B 0,C 180,E1 -978.452,E2 -978.452} C_VEL
LIN {X 0,Y 594.53,Z 348.312,A -85,B 0,C 180,E1 -978.92,E2 -978.92} C_VEL
LIN {X 0,Y 594.471,Z 360.517,A -85,B 0,C 180,E1 -979.527,E2 -979.527} C_VEL
LIN {X 0,Y 594.45,Z 371.313,A -85,B 0,C 180,E1 -980.215,E2 -980.215} C_VEL
LIN {X 0,Y 594.404,Z 381.076,A -85,B 0,C 180,E1 -980.987,E2 -980.987} C_VEL
LIN {X 0,Y 594.366,Z 389.968,A -85,B 0,C 180,E1 -981.843,E2 -981.843} C_VEL
LIN {X 0,Y 594.345,Z 398.67,A -85,B 0,C 180,E1 -982.868,E2 -982.868} C_VEL
LIN {X 0,Y 594.29,Z 405.602,A -85,B 0,C 180,E1 -983.89,E2 -983.89} C_VEL
LIN {X 0,Y 594.253,Z 411.15,A -85,B 0,C 180,E1 -984.911,E2 -984.911} C_VEL
LIN {X 0,Y 594.263,Z 415.505,A -85,B 0,C 180,E1 -985.931,E2 -985.931} C_VEL
LIN {X 0,Y 594.267,Z 417.821,A -85,B 0,C 180,E1 -986.61,E2 -986.61} C_VEL
LIN {X 0,Y 594.225,Z 419.682,A -85,B 0,C 180,E1 -987.288,E2 -987.288} C_VEL
LIN {X 0,Y 594.242,Z 421.115,A -85,B 0,C 180,E1 -987.967,E2 -987.967} C_VEL
LIN {X 0,Y 594.247,Z 422.135,A -85,B 0,C 180,E1 -988.645,E2 -988.645} C_VEL
LIN {X 0,Y 594.236,Z 422.983,A -85,B 0,C 180,E1 -990,E2 -990} C_VEL
LIN {X 0,Y 594.239,Z 422.813,A -85,B 0,C 180,E1 -990.678,E2 -990.678} C_VEL
LIN {X 0,Y 594.248,Z 422.239,A -85,B 0,C 180,E1 -991.355,E2 -991.355} C_VEL
LIN {X 0,Y 594.226,Z 419.914,A -85,B 0,C 180,E1 -992.712,E2 -992.712} C_VEL
LIN {X 0,Y 594.289,Z 417.042,A -85,B 0,C 180,E1 -993.729,E2 -993.729} C_VEL
LIN {X 0,Y 594.242,Z 413.141,A -85,B 0,C 180,E1 -994.749,E2 -994.749} C_VEL
LIN {X 0,Y 594.3,Z 408.099,A -85,B 0,C 180,E1 -995.769,E2 -995.769} C_VEL
LIN {X 0,Y 594.316,Z 401.767,A -85,B 0,C 180,E1 -996.791,E2 -996.791} C_VEL
LIN {X 0,Y 594.346,Z 393.876,A -85,B 0,C 180,E1 -997.816,E2 -997.816} C_VEL
LIN {X 0,Y 594.381,Z 384.011,A -85,B 0,C 180,E1 -998.842,E2 -998.842} C_VEL
LIN {X 0,Y 594.431,Z 373.691,A -85,B 0,C 180,E1 -999.699,E2 -999.699} C_VEL
LIN {X 0,Y 594.466,Z 362.082,A -85,B 0,C 180,E1 -1000.473,E2 -1000.473} C_VEL
LIN {X 0,Y 594.507,Z 350.889,A -85,B 0,C 180,E1 -1001.058,E2 -1001.058} C_VEL
LIN {X 0,Y 594.589,Z 338.502,A -85,B 0,C 180,E1 -1001.548,E2 -1001.548} C_VEL
LIN {X 0,Y 594.638,Z 325.485,A -85,B 0,C 180,E1 -1001.915,E2 -1001.915} C_VEL
LIN {X 0,Y 594.485,Z 320.198,A -85,B 0,C 180,E1 -1002.026,E2 -1002.026} C_VEL
LIN {X 0,Y 594.249,Z 318.533,A -85,B 0,C 180,E1 -1002.075,E2 -1002.075} C_VEL
LIN {X 0,Y 594.256,Z 312.569,A -85,B 0,C 180,E1 -1005.081,E2 -1005.081} C_VEL
LIN {X 0,Y 594.236,Z 307.037,A -85,B 0,C 180,E1 -1007.909,E2 -1007.909} C_VEL
LIN {X 0,Y 594.3,Z 301.504,A -85,B 0,C 180,E1 -1010.779,E2 -1010.779} C_VEL
LIN {X 0,Y 594.283,Z 295.971,A -85,B 0,C 180,E1 -1013.709,E2 -1013.709} C_VEL
LIN {X 0,Y 594.296,Z 291.718,A -85,B 0,C 180,E1 -1016.004,E2 -1016.004} C_VEL
LIN {X 0,Y 594.275,Z 287.602,A -85,B 0,C 180,E1 -1018.232,E2 -1018.232} C_VEL
LIN {X 0,Y 594.322,Z 281.737,A -85,B 0,C 180,E1 -1021.353,E2 -1021.353} C_VEL
LIN {X 0,Y 594.324,Z 275.731,A -85,B 0,C 180,E1 -1024.443,E2 -1024.443} C_VEL
LIN {X 0,Y 594.336,Z 275.457,A -85,B 0,C 180,E1 -1024.583,E2 -1024.583} C_VEL
LIN {X 0,Y 594.389,Z 275.446,A -85,B 0,C 180,E1 -1027.608,E2 -1027.608} C_VEL
LIN {X 0,Y 594.361,Z 275.449,A -85,B 0,C 180,E1 -1030.568,E2 -1030.568} C_VEL
LIN {X 0,Y 594.371,Z 275.449,A -85,B 0,C 180,E1 -1033.299,E2 -1033.299} C_VEL
LIN {X 0,Y 594.363,Z 275.452,A -85,B 0,C 180,E1 -1036.161,E2 -1036.161} C_VEL
LIN {X 0,Y 594.376,Z 275.448,A -85,B 0,C 180,E1 -1038.535,E2 -1038.535} C_VEL
LIN {X 0,Y 594.379,Z 275.449,A -85,B 0,C 180,E1 -1041.297,E2 -1041.297} C_VEL
LIN {X 0,Y 594.353,Z 275.451,A -85,B 0,C 180,E1 -1043.755,E2 -1043.755} C_VEL
LIN {X 0,Y 594.322,Z 275.66,A -85,B 0,C 180,E1 -1045.557,E2 -1045.557} C_VEL
LIN {X 0,Y 594.304,Z 281.565,A -85,B 0,C 180,E1 -1048.646,E2 -1048.646} C_VEL
LIN {X 0,Y 594.264,Z 286.184,A -85,B 0,C 180,E1 -1051.064,E2 -1051.064} C_VEL
LIN {X 0,Y 594.271,Z 290.274,A -85,B 0,C 180,E1 -1053.295,E2 -1053.295} C_VEL
LIN {X 0,Y 594.281,Z 294.496,A -85,B 0,C 180,E1 -1055.59,E2 -1055.59} C_VEL
LIN {X 0,Y 594.276,Z 298.568,A -85,B 0,C 180,E1 -1057.763,E2 -1057.763} C_VEL
LIN {X 0,Y 594.244,Z 302.715,A -85,B 0,C 180,E1 -1059.942,E2 -1059.942} C_VEL
LIN {X 0,Y 594.245,Z 306.862,A -85,B 0,C 180,E1 -1062.091,E2 -1062.091} C_VEL
LIN {X 0,Y 594.252,Z 311.009,A -85,B 0,C 180,E1 -1064.216,E2 -1064.216} C_VEL
LIN {X 0,Y 594.227,Z 316.539,A -85,B 0,C 180,E1 -1067.014,E2 -1067.014} C_VEL
LIN {X 0,Y 594.262,Z 318.772,A -85,B 0,C 180,E1 -1068.034,E2 -1068.034} C_VEL
LIN {X 0,Y 594.66,Z 323.434,A -85,B 0,C 180,E1 -1068.128,E2 -1068.128} C_VEL
LIN {X 0,Y 594.592,Z 335.79,A -85,B 0,C 180,E1 -1068.452,E2 -1068.452} C_VEL
LIN {X 0,Y 594.539,Z 346.852,A -85,B 0,C 180,E1 -1068.855,E2 -1068.855} C_VEL
LIN {X 0,Y 594.482,Z 358.967,A -85,B 0,C 180,E1 -1069.441,E2 -1069.441} C_VEL
LIN {X 0,Y 594.454,Z 370.089,A -85,B 0,C 180,E1 -1070.129,E2 -1070.129} C_VEL
LIN {X 0,Y 594.406,Z 379.093,A -85,B 0,C 180,E1 -1070.815,E2 -1070.815} C_VEL
LIN {X 0,Y 594.373,Z 388.345,A -85,B 0,C 180,E1 -1071.672,E2 -1071.672} C_VEL
LIN {X 0,Y 594.317,Z 397.332,A -85,B 0,C 180,E1 -1072.697,E2 -1072.697} C_VEL
LIN {X 0,Y 594.285,Z 403.858,A -85,B 0,C 180,E1 -1073.612,E2 -1073.612} C_VEL
LIN {X 0,Y 594.289,Z 409.446,A -85,B 0,C 180,E1 -1074.571,E2 -1074.571} C_VEL
LIN {X 0,Y 594.27,Z 414.188,A -85,B 0,C 180,E1 -1075.591,E2 -1075.591} C_VEL
LIN {X 0,Y 594.267,Z 417.82,A -85,B 0,C 180,E1 -1076.61,E2 -1076.61} C_VEL
LIN {X 0,Y 594.225,Z 419.689,A -85,B 0,C 180,E1 -1077.288,E2 -1077.288} C_VEL
LIN {X 0,Y 594.242,Z 421.117,A -85,B 0,C 180,E1 -1077.967,E2 -1077.967} C_VEL
LIN {X 0,Y 594.247,Z 422.133,A -85,B 0,C 180,E1 -1078.645,E2 -1078.645} C_VEL
LIN {X 0,Y 594.24,Z 422.754,A -85,B 0,C 180,E1 -1079.322,E2 -1079.322} C_VEL
LIN {X 0,Y 594.236,Z 422.98,A -85,B 0,C 180,E1 -1080,E2 -1080} C_VEL
LIN {X 0,Y 594.239,Z 422.811,A -85,B 0,C 180,E1 -1080.678,E2 -1080.678} C_VEL
LIN {X 0,Y 594.248,Z 422.24,A -85,B 0,C 180,E1 -1081.355,E2 -1081.355} C_VEL
LIN {X 0,Y 594.226,Z 419.913,A -85,B 0,C 180,E1 -1082.712,E2 -1082.712} C_VEL
LIN {X 0,Y 594.289,Z 417.042,A -85,B 0,C 180,E1 -1083.729,E2 -1083.729} C_VEL
LIN {X 0,Y 594.242,Z 413.142,A -85,B 0,C 180,E1 -1084.749,E2 -1084.749} C_VEL
LIN {X 0,Y 594.3,Z 408.101,A -85,B 0,C 180,E1 -1085.769,E2 -1085.769} C_VEL
LIN {X 0,Y 594.316,Z 401.764,A -85,B 0,C 180,E1 -1086.791,E2 -1086.791} C_VEL
LIN {X 0,Y 594.346,Z 393.876,A -85,B 0,C 180,E1 -1087.816,E2 -1087.816} C_VEL
LIN {X 0,Y 594.381,Z 384.021,A -85,B 0,C 180,E1 -1088.842,E2 -1088.842} C_VEL
LIN {X 0,Y 594.431,Z 373.676,A -85,B 0,C 180,E1 -1089.699,E2 -1089.699} C_VEL
LIN {X 0,Y 594.453,Z 363.478,A -85,B 0,C 180,E1 -1090.387,E2 -1090.387} C_VEL
LIN {X 0,Y 594.497,Z 351.738,A -85,B 0,C 180,E1 -1091.019,E2 -1091.019} C_VEL
LIN {X 0,Y 594.578,Z 339.82,A -85,B 0,C 180,E1 -1091.505,E2 -1091.505} C_VEL
LIN {X 0,Y 594.65,Z 327.302,A -85,B 0,C 180,E1 -1091.872,E2 -1091.872} C_VEL
LIN {X 0,Y 594.485,Z 320.207,A -85,B 0,C 180,E1 -1092.026,E2 -1092.026} C_VEL
LIN {X 0,Y 594.249,Z 318.533,A -85,B 0,C 180,E1 -1092.075,E2 -1092.075} C_VEL
LIN {X 0,Y 594.256,Z 312.569,A -85,B 0,C 180,E1 -1095.081,E2 -1095.081} C_VEL
LIN {X 0,Y 594.236,Z 307.037,A -85,B 0,C 180,E1 -1097.909,E2 -1097.909} C_VEL
LIN {X 0,Y 594.3,Z 301.504,A -85,B 0,C 180,E1 -1100.779,E2 -1100.779} C_VEL
LIN {X 0,Y 594.283,Z 295.971,A -85,B 0,C 180,E1 -1103.709,E2 -1103.709} C_VEL
LIN {X 0,Y 594.296,Z 291.718,A -85,B 0,C 180,E1 -1106.004,E2 -1106.004} C_VEL
LIN {X 0,Y 594.252,Z 287.359,A -85,B 0,C 180,E1 -1108.234,E2 -1108.234} C_VEL
LIN {X 0,Y 594.258,Z 282.507,A -85,B 0,C 180,E1 -1110.567,E2 -1110.567} C_VEL
LIN {X 0,Y 594.255,Z 276.828,A -85,B 0,C 180,E1 -1112.958,E2 -1112.958} C_VEL
LIN {X 0,Y 594.295,Z 275.462,A -85,B 0,C 180,E1 -1113.563,E2 -1113.563} C_VEL
LIN {X 0,Y 594.328,Z 275.455,A -85,B 0,C 180,E1 -1115.411,E2 -1115.411} C_VEL
LIN {X 0,Y 594.381,Z 275.449,A -85,B 0,C 180,E1 -1117.941,E2 -1117.941} C_VEL
LIN {X 0,Y 594.38,Z 275.447,A -85,B 0,C 180,E1 -1120.822,E2 -1120.822} C_VEL
LIN {X 0,Y 594.37,Z 275.448,A -85,B 0,C 180,E1 -1123.839,E2 -1123.839} C_VEL
LIN {X 0,Y 594.361,Z 275.45,A -85,B 0,C 180,E1 -1126.7,E2 -1126.7} C_VEL
LIN {X 0,Y 594.369,Z 275.451,A -85,B 0,C 180,E1 -1129.433,E2 -1129.433} C_VEL
LIN {X 0,Y 594.391,Z 275.447,A -85,B 0,C 180,E1 -1132.392,E2 -1132.392} C_VEL
LIN {X 0,Y 594.362,Z 275.529,A -85,B 0,C 180,E1 -1133.756,E2 -1133.756} C_VEL
LIN {X 0,Y 594.804,Z 278.598,A -85,B 0,C 180,E1 -1134.622,E2 -1134.622} C_VEL
LIN {X 0,Y 594.653,Z 289.341,A -85,B 0,C 180,E1 -1137.469,E2 -1137.469} C_VEL
LIN {X 0,Y 594.627,Z 298.907,A -85,B 0,C 180,E1 -1139.938,E2 -1139.938} C_VEL
LIN {X 0,Y 594.572,Z 309.293,A -85,B 0,C 180,E1 -1142.549,E2 -1142.549} C_VEL
LIN {X 0,Y 594.487,Z 320.038,A -85,B 0,C 180,E1 -1145.186,E2 -1145.186} C_VEL
LIN {X 0,Y 594.457,Z 330.78,A -85,B 0,C 180,E1 -1147.77,E2 -1147.77} C_VEL
LIN {X 0,Y 594.417,Z 341.523,A -85,B 0,C 180,E1 -1150.308,E2 -1150.308} C_VEL
LIN {X 0,Y 594.384,Z 353.526,A -85,B 0,C 180,E1 -1153.097,E2 -1153.097} C_VEL
LIN {X 0,Y 594.323,Z 366.583,A -85,B 0,C 180,E1 -1156.085,E2 -1156.085} C_VEL
LIN {X 0,Y 594.293,Z 374.712,A -85,B 0,C 180,E1 -1157.926,E2 -1157.926} C_VEL
LIN {X 0,Y 594.695,Z 380.085,A -85,B 0,C 180,E1 -1158.021,E2 -1158.021} C_VEL
LIN {X 0,Y 594.63,Z 393.734,A -85,B 0,C 180,E1 -1158.344,E2 -1158.344} C_VEL
LIN {X 0,Y 594.55,Z 404.783,A -85,B 0,C 180,E1 -1158.726,E2 -1158.726} C_VEL
LIN {X 0,Y 594.488,Z 416.633,A -85,B 0,C 180,E1 -1159.269,E2 -1159.269} C_VEL
LIN {X 0,Y 594.469,Z 428.197,A -85,B 0,C 180,E1 -1159.957,E2 -1159.957} C_VEL
LIN {X 0,Y 594.414,Z 438.594,A -85,B 0,C 180,E1 -1160.73,E2 -1160.73} C_VEL
LIN {X 0,Y 594.383,Z 447.111,A -85,B 0,C 180,E1 -1161.5,E2 -1161.5} C_VEL
LIN {X 0,Y 594.347,Z 454.96,A -85,B 0,C 180,E1 -1162.355,E2 -1162.355} C_VEL
LIN {X 0,Y 594.283,Z 462.812,A -85,B 0,C 180,E1 -1163.408,E2 -1163.408} C_VEL
LIN {X 0,Y 594.289,Z 469.68,A -85,B 0,C 180,E1 -1164.571,E2 -1164.571} C_VEL
LIN {X 0,Y 594.27,Z 474.371,A -85,B 0,C 180,E1 -1165.591,E2 -1165.591} C_VEL
LIN {X 0,Y 594.267,Z 477.956,A -85,B 0,C 180,E1 -1166.61,E2 -1166.61} C_VEL
LIN {X 0,Y 594.226,Z 479.809,A -85,B 0,C 180,E1 -1167.288,E2 -1167.288} C_VEL
LIN {X 0,Y 594.242,Z 481.202,A -85,B 0,C 180,E1 -1167.967,E2 -1167.967} C_VEL
LIN {X 0,Y 594.239,Z 482.784,A -85,B 0,C 180,E1 -1169.322,E2 -1169.322} C_VEL
LIN {X 0,Y 594.236,Z 483,A -85,B 0,C 180,E1 -1170,E2 -1170} C_VEL
LIN {X 0,Y 594.247,Z 482.184,A -85,B 0,C 180,E1 -1171.355,E2 -1171.355} C_VEL
LIN {X 0,Y 594.242,Z 481.202,A -85,B 0,C 180,E1 -1172.033,E2 -1172.033} C_VEL
LIN {X 0,Y 594.226,Z 479.809,A -85,B 0,C 180,E1 -1172.712,E2 -1172.712} C_VEL
LIN {X 0,Y 594.289,Z 476.896,A -85,B 0,C 180,E1 -1173.729,E2 -1173.729} C_VEL
LIN {X 0,Y 594.241,Z 472.95,A -85,B 0,C 180,E1 -1174.749,E2 -1174.749} C_VEL
LIN {X 0,Y 594.305,Z 466.877,A -85,B 0,C 180,E1 -1175.939,E2 -1175.939} C_VEL
LIN {X 0,Y 594.308,Z 460.235,A -85,B 0,C 180,E1 -1176.962,E2 -1176.962} C_VEL
LIN {X 0,Y 594.359,Z 451.989,A -85,B 0,C 180,E1 -1177.986,E2 -1177.986} C_VEL
LIN {X 0,Y 594.382,Z 443.536,A -85,B 0,C 180,E1 -1178.842,E2 -1178.842} C_VEL
LIN {X 0,Y 594.431,Z 433.091,A -85,B 0,C 180,E1 -1179.699,E2 -1179.699} C_VEL
LIN {X 0,Y 594.454,Z 422.756,A -85,B 0,C 180,E1 -1180.387,E2 -1180.387} C_VEL
LIN {X 0,Y 594.501,Z 410.771,A -85,B 0,C 180,E1 -1181.019,E2 -1181.019} C_VEL
LIN {X 0,Y 594.56,Z 398.49,A -85,B 0,C 180,E1 -1181.505,E2 -1181.505} C_VEL
LIN {X 0,Y 594.65,Z 385.435,A -85,B 0,C 180,E1 -1181.872,E2 -1181.872} C_VEL
LIN {X 0,Y 594.57,Z 376.481,A -85,B 0,C 180,E1 -1182.041,E2 -1182.041} C_VEL
LIN {X 0,Y 594.295,Z 374.712,A -85,B 0,C 180,E1 -1182.074,E2 -1182.074} C_VEL
LIN {X 0,Y 594.304,Z 364.544,A -85,B 0,C 180,E1 -1184.379,E2 -1184.379} C_VEL
LIN {X 0,Y 594.411,Z 352.266,A -85,B 0,C 180,E1 -1187.193,E2 -1187.193} C_VEL
LIN {X 0,Y 594.45,Z 339.988,A -85,B 0,C 180,E1 -1190.051,E2 -1190.051} C_VEL
LIN {X 0,Y 594.494,Z 327.71,A -85,B 0,C 180,E1 -1192.962,E2 -1192.962} C_VEL
LIN {X 0,Y 594.535,Z 314.964,A -85,B 0,C 180,E1 -1196.052,E2 -1196.052} C_VEL
LIN {X 0,Y 594.581,Z 304.689,A -85,B 0,C 180,E1 -1198.602,E2 -1198.602} C_VEL
LIN {X 0,Y 594.678,Z 293.946,A -85,B 0,C 180,E1 -1201.332,E2 -1201.332} C_VEL
LIN {X 0,Y 594.717,Z 283.059,A -85,B 0,C 180,E1 -1204.186,E2 -1204.186} C_VEL
LIN {X 0,Y 594.644,Z 277.065,A -85,B 0,C 180,E1 -1205.805,E2 -1205.805} C_VEL
LIN {X 0,Y 594.334,Z 275.455,A -85,B 0,C 180,E1 -1206.333,E2 -1206.333} C_VEL
LIN {X 0,Y 594.365,Z 275.452,A -85,B 0,C 180,E1 -1208.807,E2 -1208.807} C_VEL
LIN {X 0,Y 594.364,Z 275.445,A -85,B 0,C 180,E1 -1211.846,E2 -1211.846} C_VEL
LIN {X 0,Y 594.339,Z 275.453,A -85,B 0,C 180,E1 -1214.806,E2 -1214.806} C_VEL
LIN {X 0,Y 594.346,Z 275.446,A -85,B 0,C 180,E1 -1217.622,E2 -1217.622} C_VEL
LIN {X 0,Y 594.397,Z 275.449,A -85,B 0,C 180,E1 -1220.321,E2 -1220.321} C_VEL
LIN {X 0,Y 594.384,Z 275.442,A -85,B 0,C 180,E1 -1222.913,E2 -1222.913} C_VEL
LIN {X 0,Y 594.382,Z 275.45,A -85,B 0,C 180,E1 -1225.862,E2 -1225.862} C_VEL
LIN {X 0,Y 594.372,Z 275.443,A -85,B 0,C 180,E1 -1228.65,E2 -1228.65} C_VEL
LIN {X 0,Y 594.387,Z 275.443,A -85,B 0,C 180,E1 -1231.042,E2 -1231.042} C_VEL
LIN {X 0,Y 594.384,Z 275.444,A -85,B 0,C 180,E1 -1233.978,E2 -1233.978} C_VEL
LIN {X 0,Y 594.235,Z 275.469,A -85,B 0,C 180,E1 -1236.289,E2 -1236.289} C_VEL
LIN {X 0,Y 594.29,Z 278.932,A -85,B 0,C 180,E1 -1239.22,E2 -1239.22} C_VEL
LIN {X 0,Y 594.199,Z 282.448,A -85,B 0,C 180,E1 -1242.09,E2 -1242.09} C_VEL
LIN {X 0,Y 594.213,Z 285.964,A -85,B 0,C 180,E1 -1244.918,E2 -1244.918} C_VEL
LIN {X 0,Y 594.218,Z 288.6,A -85,B 0,C 180,E1 -1247.014,E2 -1247.014} C_VEL
LIN {X 0,Y 594.248,Z 290.034,A -85,B 0,C 180,E1 -1248.055,E2 -1248.055} C_VEL
LIN {X 0,Y 594.665,Z 295.388,A -85,B 0,C 180,E1 -1248.172,E2 -1248.172} C_VEL
LIN {X 0,Y 594.567,Z 309.772,A -85,B 0,C 180,E1 -1248.582,E2 -1248.582} C_VEL
LIN {X 0,Y 594.502,Z 322.227,A -85,B 0,C 180,E1 -1249.097,E2 -1249.097} C_VEL
LIN {X 0,Y 594.455,Z 333.43,A -85,B 0,C 180,E1 -1249.699,E2 -1249.699} C_VEL
LIN {X 0,Y 594.422,Z 344.811,A -85,B 0,C 180,E1 -1250.472,E2 -1250.472} C_VEL
LIN {X 0,Y 594.378,Z 354.854,A -85,B 0,C 180,E1 -1251.329,E2 -1251.329} C_VEL
LIN {X 0,Y 594.346,Z 363.067,A -85,B 0,C 180,E1 -1252.184,E2 -1252.184} C_VEL
LIN {X 0,Y 594.318,Z 371.136,A -85,B 0,C 180,E1 -1253.209,E2 -1253.209} C_VEL
LIN {X 0,Y 594.303,Z 377.615,A -85,B 0,C 180,E1 -1254.231,E2 -1254.231} C_VEL
LIN {X 0,Y 594.24,Z 382.754,A -85,B 0,C 180,E1 -1255.251,E2 -1255.251} C_VEL
LIN {X 0,Y 594.289,Z 386.743,A -85,B 0,C 180,E1 -1256.271,E2 -1256.271} C_VEL
LIN {X 0,Y 594.225,Z 389.697,A -85,B 0,C 180,E1 -1257.288,E2 -1257.288} C_VEL
LIN {X 0,Y 594.242,Z 391.132,A -85,B 0,C 180,E1 -1257.967,E2 -1257.967} C_VEL
LIN {X 0,Y 594.24,Z 392.755,A -85,B 0,C 180,E1 -1259.322,E2 -1259.322} C_VEL
LIN {X 0,Y 594.236,Z 392.996,A -85,B 0,C 180,E1 -1260,E2 -1260} C_VEL
LIN {X 0,Y 594.239,Z 392.814,A -85,B 0,C 180,E1 -1260.678,E2 -1260.678} C_VEL
LIN {X 0,Y 594.242,Z 391.277,A -85,B 0,C 180,E1 -1262.033,E2 -1262.033} C_VEL
LIN {X 0,Y 594.226,Z 389.9,A -85,B 0,C 180,E1 -1262.712,E2 -1262.712} C_VEL
LIN {X 0,Y 594.289,Z 387.026,A -85,B 0,C 180,E1 -1263.729,E2 -1263.729} C_VEL
LIN {X 0,Y 594.241,Z 383.132,A -85,B 0,C 180,E1 -1264.749,E2 -1264.749} C_VEL
LIN {X 0,Y 594.3,Z 378.106,A -85,B 0,C 180,E1 -1265.769,E2 -1265.769} C_VEL
LIN {X 0,Y 594.316,Z 371.786,A -85,B 0,C 180,E1 -1266.791,E2 -1266.791} C_VEL
LIN {X 0,Y 594.346,Z 363.856,A -85,B 0,C 180,E1 -1267.816,E2 -1267.816} C_VEL
LIN {X 0,Y 594.366,Z 355.781,A -85,B 0,C 180,E1 -1268.671,E2 -1268.671} C_VEL
LIN {X 0,Y 594.416,Z 345.949,A -85,B 0,C 180,E1 -1269.528,E2 -1269.528} C_VEL
LIN {X 0,Y 594.449,Z 334.91,A -85,B 0,C 180,E1 -1270.301,E2 -1270.301} C_VEL
LIN {X 0,Y 594.476,Z 324.084,A -85,B 0,C 180,E1 -1270.904,E2 -1270.904} C_VEL
LIN {X 0,Y 594.551,Z 311.818,A -85,B 0,C 180,E1 -1271.432,E2 -1271.432} C_VEL
LIN {X 0,Y 594.63,Z 299.721,A -85,B 0,C 180,E1 -1271.813,E2 -1271.813} C_VEL
LIN {X 0,Y 594.24,Z 296.413,A -85,B 0,C 180,E1 -1271.974,E2 -1271.974} C_VEL
LIN {X 0,Y 593.337,Z 293.757,A -85,B 0,C 180,E1 -1272.219,E2 -1272.219} C_VEL
LIN {X 0,Y 591.503,Z 290.873,A -85,B 0,C 180,E1 -1272.679,E2 -1272.679} C_VEL
LIN {X 0,Y 589.502,Z 289.072,A -85,B 0,C 180,E1 -1273.223,E2 -1273.223} C_VEL
LIN {X 0,Y 587.465,Z 287.643,A -85,B 0,C 180,E1 -1274.015,E2 -1274.015} C_VEL
LIN {X 0,Y 587.112,Z 287.121,A -85,B 0,C 180,E1 -1274.425,E2 -1274.425} C_VEL
LIN {X 0,Y 587.124,Z 284.262,A -85,B 0,C 180,E1 -1276.74,E2 -1276.74} C_VEL
LIN {X 0,Y 587.107,Z 280.799,A -85,B 0,C 180,E1 -1279.583,E2 -1279.583} C_VEL
LIN {X 0,Y 587.133,Z 278.161,A -85,B 0,C 180,E1 -1281.782,E2 -1281.782} C_VEL
LIN {X 0,Y 587.118,Z 276.402,A -85,B 0,C 180,E1 -1283.267,E2 -1283.267} C_VEL
LIN {X 0,Y 587.328,Z 276.319,A -85,B 0,C 180,E1 -1285.517,E2 -1285.517} C_VEL
LIN {X 0,Y 587.343,Z 276.318,A -85,B 0,C 180,E1 -1287.818,E2 -1287.818} C_VEL
LIN {X 0,Y 587.329,Z 276.329,A -85,B 0,C 180,E1 -1290.508,E2 -1290.508} C_VEL
LIN {X 0,Y 587.341,Z 276.319,A -85,B 0,C 180,E1 -1293.112,E2 -1293.112} C_VEL
LIN {X 0,Y 587.299,Z 276.323,A -85,B 0,C 180,E1 -1295.537,E2 -1295.537} C_VEL
LIN {X 0,Y 587.345,Z 276.322,A -85,B 0,C 180,E1 -1297.839,E2 -1297.839} C_VEL
LIN {X 0,Y 587.316,Z 276.329,A -85,B 0,C 180,E1 -1300.254,E2 -1300.254} C_VEL
LIN {X 0,Y 587.318,Z 276.321,A -85,B 0,C 180,E1 -1303.118,E2 -1303.118} C_VEL
LIN {X 0,Y 587.327,Z 276.327,A -85,B 0,C 180,E1 -1306.05,E2 -1306.05} C_VEL
LIN {X 0,Y 587.339,Z 276.319,A -85,B 0,C 180,E1 -1308.925,E2 -1308.925} C_VEL
LIN {X 0,Y 587.331,Z 276.327,A -85,B 0,C 180,E1 -1311.52,E2 -1311.52} C_VEL
LIN {X 0,Y 587.292,Z 276.327,A -85,B 0,C 180,E1 -1314.1,E2 -1314.1} C_VEL
LIN {X 0,Y 587.269,Z 276.505,A -85,B 0,C 180,E1 -1315.664,E2 -1315.664} C_VEL
LIN {X 0,Y 587.242,Z 281.429,A -85,B 0,C 180,E1 -1318.225,E2 -1318.225} C_VEL
LIN {X 0,Y 587.171,Z 286.432,A -85,B 0,C 180,E1 -1320.899,E2 -1320.899} C_VEL
LIN {X 0,Y 587.216,Z 291.648,A -85,B 0,C 180,E1 -1323.715,E2 -1323.715} C_VEL
LIN {X 0,Y 587.2,Z 295.804,A -85,B 0,C 180,E1 -1325.987,E2 -1325.987} C_VEL
LIN {X 0,Y 587.187,Z 299.951,A -85,B 0,C 180,E1 -1328.22,E2 -1328.22} C_VEL
LIN {X 0,Y 587.203,Z 305.481,A -85,B 0,C 180,E1 -1331.146,E2 -1331.146} C_VEL
LIN {X 0,Y 587.165,Z 311.01,A -85,B 0,C 180,E1 -1334.02,E2 -1334.02} C_VEL
LIN {X 0,Y 587.176,Z 315.158,A -85,B 0,C 180,E1 -1336.15,E2 -1336.15} C_VEL
LIN {X 0,Y 587.188,Z 318.72,A -85,B 0,C 180,E1 -1337.888,E2 -1337.888} C_VEL
LIN {X 0,Y 587.72,Z 324.438,A -85,B 0,C 180,E1 -1338.008,E2 -1338.008} C_VEL
LIN {X 0,Y 587.627,Z 337.296,A -85,B 0,C 180,E1 -1338.364,E2 -1338.364} C_VEL
LIN {X 0,Y 587.561,Z 348.659,A -85,B 0,C 180,E1 -1338.802,E2 -1338.802} C_VEL
LIN {X 0,Y 587.488,Z 360.526,A -85,B 0,C 180,E1 -1339.401,E2 -1339.401} C_VEL
LIN {X 0,Y 587.437,Z 371.318,A -85,B 0,C 180,E1 -1340.097,E2 -1340.097} C_VEL
LIN {X 0,Y 587.357,Z 381.077,A -85,B 0,C 180,E1 -1340.878,E2 -1340.878} C_VEL
LIN {X 0,Y 587.302,Z 389.965,A -85,B 0,C 180,E1 -1341.744,E2 -1341.744} C_VEL
LIN {X 0,Y 587.259,Z 397.318,A -85,B 0,C 180,E1 -1342.608,E2 -1342.608} C_VEL
LIN {X 0,Y 587.199,Z 404.435,A -85,B 0,C 180,E1 -1343.624,E2 -1343.624} C_VEL
LIN {X 0,Y 587.211,Z 409.445,A -85,B 0,C 180,E1 -1344.506,E2 -1344.506} C_VEL
LIN {X 0,Y 587.188,Z 414.191,A -85,B 0,C 180,E1 -1345.538,E2 -1345.538} C_VEL
LIN {X 0,Y 587.194,Z 417.826,A -85,B 0,C 180,E1 -1346.569,E2 -1346.569} C_VEL
LIN {X 0,Y 587.131,Z 419.679,A -85,B 0,C 180,E1 -1347.256,E2 -1347.256} C_VEL
LIN {X 0,Y 587.141,Z 421.109,A -85,B 0,C 180,E1 -1347.942,E2 -1347.942} C_VEL
LIN {X 0,Y 587.147,Z 422.138,A -85,B 0,C 180,E1 -1348.628,E2 -1348.628} C_VEL
LIN {X 0,Y 587.137,Z 422.975,A -85,B 0,C 180,E1 -1350,E2 -1350} C_VEL
LIN {X 0,Y 587.14,Z 422.813,A -85,B 0,C 180,E1 -1350.686,E2 -1350.686} C_VEL
LIN {X 0,Y 587.148,Z 422.24,A -85,B 0,C 180,E1 -1351.372,E2 -1351.372} C_VEL
LIN {X 0,Y 587.133,Z 419.91,A -85,B 0,C 180,E1 -1352.744,E2 -1352.744} C_VEL
LIN {X 0,Y 587.213,Z 417.038,A -85,B 0,C 180,E1 -1353.774,E2 -1353.774} C_VEL
LIN {X 0,Y 587.147,Z 413.135,A -85,B 0,C 180,E1 -1354.806,E2 -1354.806} C_VEL
LIN {X 0,Y 587.23,Z 408.087,A -85,B 0,C 180,E1 -1355.839,E2 -1355.839} C_VEL
LIN {X 0,Y 587.229,Z 401.754,A -85,B 0,C 180,E1 -1356.874,E2 -1356.874} C_VEL
LIN {X 0,Y 587.288,Z 393.875,A -85,B 0,C 180,E1 -1357.91,E2 -1357.91} C_VEL
LIN {X 0,Y 587.343,Z 383.995,A -85,B 0,C 180,E1 -1358.949,E2 -1358.949} C_VEL
LIN {X 0,Y 587.397,Z 374.813,A -85,B 0,C 180,E1 -1359.73,E2 -1359.73} C_VEL
LIN {X 0,Y 587.45,Z 364.887,A -85,B 0,C 180,E1 -1360.425,E2 -1360.425} C_VEL
LIN {X 0,Y 587.523,Z 353.063,A -85,B 0,C 180,E1 -1361.085,E2 -1361.085} C_VEL
LIN {X 0,Y 587.611,Z 340.971,A -85,B 0,C 180,E1 -1361.602,E2 -1361.602} C_VEL
LIN {X 0,Y 587.692,Z 329.023,A -85,B 0,C 180,E1 -1361.971,E2 -1361.971} C_VEL
LIN {X 0,Y 587.516,Z 321.033,A -85,B 0,C 180,E1 -1362.155,E2 -1362.155} C_VEL
LIN {X 0,Y 587.15,Z 318.532,A -85,B 0,C 180,E1 -1362.223,E2 -1362.223} C_VEL
LIN {X 0,Y 587.178,Z 313.951,A -85,B 0,C 180,E1 -1364.558,E2 -1364.558} C_VEL
LIN {X 0,Y 587.145,Z 308.419,A -85,B 0,C 180,E1 -1367.412,E2 -1367.412} C_VEL
LIN {X 0,Y 587.189,Z 304.269,A -85,B 0,C 180,E1 -1369.58,E2 -1369.58} C_VEL
LIN {X 0,Y 587.19,Z 300.12,A -85,B 0,C 180,E1 -1371.78,E2 -1371.78} C_VEL
LIN {X 0,Y 587.207,Z 294.985,A -85,B 0,C 180,E1 -1374.548,E2 -1374.548} C_VEL
LIN {X 0,Y 587.208,Z 290.425,A -85,B 0,C 180,E1 -1377.052,E2 -1377.052} C_VEL
LIN {X 0,Y 587.237,Z 284.628,A -85,B 0,C 180,E1 -1380.176,E2 -1380.176} C_VEL
LIN {X 0,Y 587.241,Z 279.126,A -85,B 0,C 180,E1 -1383.096,E2 -1383.096} C_VEL
LIN {X 0,Y 587.291,Z 276.334,A -85,B 0,C 180,E1 -1384.569,E2 -1384.569} C_VEL
LIN {X 0,Y 587.344,Z 276.324,A -85,B 0,C 180,E1 -1387.608,E2 -1387.608} C_VEL
LIN {X 0,Y 587.316,Z 276.327,A -85,B 0,C 180,E1 -1390.254,E2 -1390.254} C_VEL
LIN {X 0,Y 587.32,Z 276.326,A -85,B 0,C 180,E1 -1393.118,E2 -1393.118} C_VEL
LIN {X 0,Y 587.316,Z 276.329,A -85,B 0,C 180,E1 -1396.048,E2 -1396.048} C_VEL
LIN {X 0,Y 587.335,Z 276.328,A -85,B 0,C 180,E1 -1398.926,E2 -1398.926} C_VEL
LIN {X 0,Y 587.325,Z 276.329,A -85,B 0,C 180,E1 -1401.52,E2 -1401.52} C_VEL
LIN {X 0,Y 587.301,Z 276.329,A -85,B 0,C 180,E1 -1404.462,E2 -1404.462} C_VEL
LIN {X 0,Y 587.271,Z 276.532,A -85,B 0,C 180,E1 -1405.664,E2 -1405.664} C_VEL
LIN {X 0,Y 587.225,Z 281.419,A -85,B 0,C 180,E1 -1408.224,E2 -1408.224} C_VEL
LIN {X 0,Y 587.205,Z 286.514,A -85,B 0,C 180,E1 -1410.893,E2 -1410.893} C_VEL
LIN {X 0,Y 587.219,Z 291.874,A -85,B 0,C 180,E1 -1413.848,E2 -1413.848} C_VEL
LIN {X 0,Y 587.198,Z 297.187,A -85,B 0,C 180,E1 -1416.736,E2 -1416.736} C_VEL
LIN {X 0,Y 587.179,Z 302.716,A -85,B 0,C 180,E1 -1419.69,E2 -1419.69} C_VEL
LIN {X 0,Y 587.155,Z 306.863,A -85,B 0,C 180,E1 -1421.868,E2 -1421.868} C_VEL
LIN {X 0,Y 587.163,Z 312.393,A -85,B 0,C 180,E1 -1424.732,E2 -1424.732} C_VEL
LIN {X 0,Y 587.153,Z 317.923,A -85,B 0,C 180,E1 -1427.558,E2 -1427.558} C_VEL
LIN {X 0,Y 587.188,Z 318.762,A -85,B 0,C 180,E1 -1427.888,E2 -1427.888} C_VEL
LIN {X 0,Y 587.738,Z 323.458,A -85,B 0,C 180,E1 -1427.987,E2 -1427.987} C_VEL
LIN {X 0,Y 587.632,Z 335.74,A -85,B 0,C 180,E1 -1428.312,E2 -1428.312} C_VEL
LIN {X 0,Y 587.566,Z 347.791,A -85,B 0,C 180,E1 -1428.761,E2 -1428.761} C_VEL
LIN {X 0,Y 587.488,Z 360.542,A -85,B 0,C 180,E1 -1429.401,E2 -1429.401} C_VEL
LIN {X 0,Y 587.439,Z 371.281,A -85,B 0,C 180,E1 -1430.097,E2 -1430.097} C_VEL
LIN {X 0,Y 587.357,Z 381.08,A -85,B 0,C 180,E1 -1430.878,E2 -1430.878} C_VEL
LIN {X 0,Y 587.303,Z 389.987,A -85,B 0,C 180,E1 -1431.744,E2 -1431.744} C_VEL
LIN {X 0,Y 587.274,Z 398.674,A -85,B 0,C 180,E1 -1432.781,E2 -1432.781} C_VEL
LIN {X 0,Y 587.214,Z 405.594,A -85,B 0,C 180,E1 -1433.816,E2 -1433.816} C_VEL
LIN {X 0,Y 587.167,Z 411.138,A -85,B 0,C 180,E1 -1434.85,E2 -1434.85} C_VEL
LIN {X 0,Y 587.182,Z 415.498,A -85,B 0,C 180,E1 -1435.882,E2 -1435.882} C_VEL
LIN {X 0,Y 587.194,Z 417.824,A -85,B 0,C 180,E1 -1436.569,E2 -1436.569} C_VEL
LIN {X 0,Y 587.131,Z 419.689,A -85,B 0,C 180,E1 -1437.256,E2 -1437.256} C_VEL
LIN {X 0,Y 587.141,Z 421.11,A -85,B 0,C 180,E1 -1437.942,E2 -1437.942} C_VEL
LIN {X 0,Y 587.147,Z 422.134,A -85,B 0,C 180,E1 -1438.628,E2 -1438.628} C_VEL
LIN {X 0,Y 587.14,Z 422.755,A -85,B 0,C 180,E1 -1439.314,E2 -1439.314} C_VEL
LIN {X 0,Y 587.14,Z 422.809,A -85,B 0,C 180,E1 -1440.686,E2 -1440.686} C_VEL
LIN {X 0,Y 587.148,Z 422.241,A -85,B 0,C 180,E1 -1441.372,E2 -1441.372} C_VEL
LIN {X 0,Y 587.133,Z 419.908,A -85,B 0,C 180,E1 -1442.744,E2 -1442.744} C_VEL
LIN {X 0,Y 587.213,Z 417.038,A -85,B 0,C 180,E1 -1443.774,E2 -1443.774} C_VEL
LIN {X 0,Y 587.147,Z 413.136,A -85,B 0,C 180,E1 -1444.806,E2 -1444.806} C_VEL
LIN {X 0,Y 587.23,Z 408.089,A -85,B 0,C 180,E1 -1445.839,E2 -1445.839} C_VEL
LIN {X 0,Y 587.229,Z 401.751,A -85,B 0,C 180,E1 -1446.874,E2 -1446.874} C_VEL
LIN {X 0,Y 587.288,Z 393.874,A -85,B 0,C 180,E1 -1447.91,E2 -1447.91} C_VEL
LIN {X 0,Y 587.331,Z 384.01,A -85,B 0,C 180,E1 -1448.949,E2 -1448.949} C_VEL
LIN {X 0,Y 587.425,Z 374.814,A -85,B 0,C 180,E1 -1449.729,E2 -1449.729} C_VEL
LIN {X 0,Y 587.454,Z 364.861,A -85,B 0,C 180,E1 -1450.425,E2 -1450.425} C_VEL
LIN {X 0,Y 587.518,Z 354.067,A -85,B 0,C 180,E1 -1451.034,E2 -1451.034} C_VEL
LIN {X 0,Y 587.601,Z 341.349,A -85,B 0,C 180,E1 -1451.589,E2 -1451.589} C_VEL
LIN {X 0,Y 587.692,Z 329.044,A -85,B 0,C 180,E1 -1451.97,E2 -1451.97} C_VEL
LIN {X 0,Y 587.521,Z 320.902,A -85,B 0,C 180,E1 -1452.157,E2 -1452.157} C_VEL
LIN {X 0,Y 587.15,Z 318.532,A -85,B 0,C 180,E1 -1452.223,E2 -1452.223} C_VEL
LIN {X 0,Y 587.178,Z 313.951,A -85,B 0,C 180,E1 -1454.558,E2 -1454.558} C_VEL
LIN {X 0,Y 587.145,Z 308.419,A -85,B 0,C 180,E1 -1457.412,E2 -1457.412} C_VEL
LIN {X 0,Y 587.189,Z 304.269,A -85,B 0,C 180,E1 -1459.58,E2 -1459.58} C_VEL
LIN {X 0,Y 587.19,Z 300.12,A -85,B 0,C 180,E1 -1461.78,E2 -1461.78} C_VEL
LIN {X 0,Y 587.207,Z 294.985,A -85,B 0,C 180,E1 -1464.548,E2 -1464.548} C_VEL
LIN {X 0,Y 587.187,Z 290.256,A -85,B 0,C 180,E1 -1467.053,E2 -1467.053} C_VEL
LIN {X 0,Y 587.166,Z 283.736,A -85,B 0,C 180,E1 -1470.18,E2 -1470.18} C_VEL
LIN {X 0,Y 587.147,Z 278.068,A -85,B 0,C 180,E1 -1472.591,E2 -1472.591} C_VEL
LIN {X 0,Y 587.17,Z 276.349,A -85,B 0,C 180,E1 -1473.314,E2 -1473.314} C_VEL
LIN {X 0,Y 587.309,Z 276.332,A -85,B 0,C 180,E1 -1475.057,E2 -1475.057} C_VEL
LIN {X 0,Y 587.337,Z 276.328,A -85,B 0,C 180,E1 -1477.838,E2 -1477.838} C_VEL
LIN {X 0,Y 587.313,Z 276.33,A -85,B 0,C 180,E1 -1480.255,E2 -1480.255} C_VEL
LIN {X 0,Y 587.306,Z 276.331,A -85,B 0,C 180,E1 -1483.117,E2 -1483.117} C_VEL
LIN {X 0,Y 587.325,Z 276.326,A -85,B 0,C 180,E1 -1486.049,E2 -1486.049} C_VEL
LIN {X 0,Y 587.339,Z 276.324,A -85,B 0,C 180,E1 -1488.925,E2 -1488.925} C_VEL
LIN {X 0,Y 587.322,Z 276.326,A -85,B 0,C 180,E1 -1491.52,E2 -1491.52} C_VEL
LIN {X 0,Y 587.347,Z 276.488,A -85,B 0,C 180,E1 -1493.52,E2 -1493.52} C_VEL
LIN {X 0,Y 587.895,Z 280.586,A -85,B 0,C 180,E1 -1494.688,E2 -1494.688} C_VEL
LIN {X 0,Y 587.736,Z 290.876,A -85,B 0,C 180,E1 -1497.446,E2 -1497.446} C_VEL
LIN {X 0,Y 587.669,Z 300.085,A -85,B 0,C 180,E1 -1499.849,E2 -1499.849} C_VEL
LIN {X 0,Y 587.593,Z 310.948,A -85,B 0,C 180,E1 -1502.612,E2 -1502.612} C_VEL
LIN {X 0,Y 587.498,Z 322.147,A -85,B 0,C 180,E1 -1505.389,E2 -1505.389} C_VEL
LIN {X 0,Y 587.444,Z 332.314,A -85,B 0,C 180,E1 -1507.861,E2 -1507.861} C_VEL
LIN {X 0,Y 587.38,Z 344.364,A -85,B 0,C 180,E1 -1510.735,E2 -1510.735} C_VEL
LIN {X 0,Y 587.313,Z 355.336,A -85,B 0,C 180,E1 -1513.31,E2 -1513.31} C_VEL
LIN {X 0,Y 587.256,Z 367.614,A -85,B 0,C 180,E1 -1516.152,E2 -1516.152} C_VEL
LIN {X 0,Y 587.239,Z 374.712,A -85,B 0,C 180,E1 -1517.779,E2 -1517.779} C_VEL
LIN {X 0,Y 587.756,Z 380.085,A -85,B 0,C 180,E1 -1517.878,E2 -1517.878} C_VEL
LIN {X 0,Y 587.664,Z 393.734,A -85,B 0,C 180,E1 -1518.204,E2 -1518.204} C_VEL
LIN {X 0,Y 587.564,Z 406.422,A -85,B 0,C 180,E1 -1518.657,E2 -1518.657} C_VEL
LIN {X 0,Y 587.477,Z 418.207,A -85,B 0,C 180,E1 -1519.227,E2 -1519.227} C_VEL
LIN {X 0,Y 587.462,Z 429.475,A -85,B 0,C 180,E1 -1519.923,E2 -1519.923} C_VEL
LIN {X 0,Y 587.384,Z 439.646,A -85,B 0,C 180,E1 -1520.704,E2 -1520.704} C_VEL
LIN {X 0,Y 587.34,Z 448.787,A -85,B 0,C 180,E1 -1521.571,E2 -1521.571} C_VEL
LIN {X 0,Y 587.259,Z 457.691,A -85,B 0,C 180,E1 -1522.608,E2 -1522.608} C_VEL
LIN {X 0,Y 587.195,Z 464.745,A -85,B 0,C 180,E1 -1523.627,E2 -1523.627} C_VEL
LIN {X 0,Y 587.211,Z 469.68,A -85,B 0,C 180,E1 -1524.506,E2 -1524.506} C_VEL
LIN {X 0,Y 587.188,Z 474.371,A -85,B 0,C 180,E1 -1525.538,E2 -1525.538} C_VEL
LIN {X 0,Y 587.193,Z 477.956,A -85,B 0,C 180,E1 -1526.569,E2 -1526.569} C_VEL
LIN {X 0,Y 587.132,Z 479.809,A -85,B 0,C 180,E1 -1527.256,E2 -1527.256} C_VEL
LIN {X 0,Y 587.141,Z 481.202,A -85,B 0,C 180,E1 -1527.942,E2 -1527.942} C_VEL
LIN {X 0,Y 587.14,Z 482.784,A -85,B 0,C 180,E1 -1529.314,E2 -1529.314} C_VEL
LIN {X 0,Y 587.137,Z 483,A -85,B 0,C 180,E1 -1530,E2 -1530} C_VEL
LIN {X 0,Y 587.147,Z 482.185,A -85,B 0,C 180,E1 -1531.372,E2 -1531.372} C_VEL
LIN {X 0,Y 587.141,Z 481.202,A -85,B 0,C 180,E1 -1532.058,E2 -1532.058} C_VEL
LIN {X 0,Y 587.132,Z 479.809,A -85,B 0,C 180,E1 -1532.744,E2 -1532.744} C_VEL
LIN {X 0,Y 587.213,Z 476.896,A -85,B 0,C 180,E1 -1533.774,E2 -1533.774} C_VEL
LIN {X 0,Y 587.147,Z 472.95,A -85,B 0,C 180,E1 -1534.806,E2 -1534.806} C_VEL
LIN {X 0,Y 587.218,Z 466.877,A -85,B 0,C 180,E1 -1536.011,E2 -1536.011} C_VEL
LIN {X 0,Y 587.245,Z 460.235,A -85,B 0,C 180,E1 -1537.046,E2 -1537.046} C_VEL
LIN {X 0,Y 587.299,Z 451.989,A -85,B 0,C 180,E1 -1538.083,E2 -1538.083} C_VEL
LIN {X 0,Y 587.343,Z 443.536,A -85,B 0,C 180,E1 -1538.949,E2 -1538.949} C_VEL
LIN {X 0,Y 587.416,Z 433.092,A -85,B 0,C 180,E1 -1539.816,E2 -1539.816} C_VEL
LIN {X 0,Y 587.472,Z 422.757,A -85,B 0,C 180,E1 -1540.512,E2 -1540.512} C_VEL
LIN {X 0,Y 587.53,Z 411.162,A -85,B 0,C 180,E1 -1541.133,E2 -1541.133} C_VEL
LIN {X 0,Y 587.594,Z 398.692,A -85,B 0,C 180,E1 -1541.637,E2 -1541.637} C_VEL
LIN {X 0,Y 587.717,Z 385.435,A -85,B 0,C 180,E1 -1542.014,E2 -1542.014} C_VEL
LIN {X 0,Y 587.548,Z 376.858,A -85,B 0,C 180,E1 -1542.182,E2 -1542.182} C_VEL
LIN {X 0,Y 587.24,Z 374.712,A -85,B 0,C 180,E1 -1542.221,E2 -1542.221} C_VEL
LIN {X 0,Y 587.275,Z 363.009,A -85,B 0,C 180,E1 -1544.91,E2 -1544.91} C_VEL
LIN {X 0,Y 587.345,Z 350.731,A -85,B 0,C 180,E1 -1547.766,E2 -1547.766} C_VEL
LIN {X 0,Y 587.41,Z 338.453,A -85,B 0,C 180,E1 -1550.668,E2 -1550.668} C_VEL
LIN {X 0,Y 587.486,Z 326.175,A -85,B 0,C 180,E1 -1553.626,E2 -1553.626} C_VEL
LIN {X 0,Y 587.577,Z 313.897,A -85,B 0,C 180,E1 -1556.65,E2 -1556.65} C_VEL
LIN {X 0,Y 587.671,Z 303.154,A -85,B 0,C 180,E1 -1559.362,E2 -1559.362} C_VEL
LIN {X 0,Y 587.752,Z 292.279,A -85,B 0,C 180,E1 -1562.183,E2 -1562.183} C_VEL
LIN {X 0,Y 587.809,Z 282.953,A -85,B 0,C 180,E1 -1564.673,E2 -1564.673} C_VEL
LIN {X 0,Y 587.731,Z 278.598,A -85,B 0,C 180,E1 -1565.869,E2 -1565.869} C_VEL
LIN {X 0,Y 587.307,Z 276.331,A -85,B 0,C 180,E1 -1566.537,E2 -1566.537} C_VEL
LIN {X 0,Y 587.318,Z 276.326,A -85,B 0,C 180,E1 -1569.362,E2 -1569.362} C_VEL
LIN {X 0,Y 587.304,Z 276.326,A -85,B 0,C 180,E1 -1572.104,E2 -1572.104} C_VEL
LIN {X 0,Y 587.292,Z 276.328,A -85,B 0,C 180,E1 -1575.086,E2 -1575.086} C_VEL
LIN {X 0,Y 587.311,Z 276.325,A -85,B 0,C 180,E1 -1577.924,E2 -1577.924} C_VEL
LIN {X 0,Y 587.348,Z 276.322,A -85,B 0,C 180,E1 -1580.641,E2 -1580.641} C_VEL
LIN {X 0,Y 587.35,Z 276.318,A -85,B 0,C 180,E1 -1583.293,E2 -1583.293} C_VEL
LIN {X 0,Y 587.361,Z 276.323,A -85,B 0,C 180,E1 -1585.78,E2 -1585.78} C_VEL
LIN {X 0,Y 587.343,Z 276.322,A -85,B 0,C 180,E1 -1588.231,E2 -1588.231} C_VEL
LIN {X 0,Y 587.353,Z 276.318,A -85,B 0,C 180,E1 -1590.867,E2 -1590.867} C_VEL
LIN {X 0,Y 587.361,Z 276.321,A -85,B 0,C 180,E1 -1593.819,E2 -1593.819} C_VEL
LIN {X 0,Y 587.217,Z 276.341,A -85,B 0,C 180,E1 -1595.988,E2 -1595.988} C_VEL
LIN {X 0,Y 587.151,Z 276.349,A -85,B 0,C 180,E1 -1596.734,E2 -1596.734} C_VEL
LIN {X 0,Y 587.159,Z 279.812,A -85,B 0,C 180,E1 -1599.689,E2 -1599.689} C_VEL
LIN {X 0,Y 587.122,Z 283.328,A -85,B 0,C 180,E1 -1602.587,E2 -1602.587} C_VEL
LIN {X 0,Y 587.13,Z 285.964,A -85,B 0,C 180,E1 -1604.732,E2 -1604.732} C_VEL
LIN {X 0,Y 587.122,Z 288.601,A -85,B 0,C 180,E1 -1606.854,E2 -1606.854} C_VEL
LIN {X 0,Y 587.162,Z 290.076,A -85,B 0,C 180,E1 -1607.909,E2 -1607.909} C_VEL
LIN {X 0,Y 587.725,Z 295.403,A -85,B 0,C 180,E1 -1608.03,E2 -1608.03} C_VEL
LIN {X 0,Y 587.59,Z 308.797,A -85,B 0,C 180,E1 -1608.411,E2 -1608.411} C_VEL
LIN {X 0,Y 587.52,Z 321.196,A -85,B 0,C 180,E1 -1608.916,E2 -1608.916} C_VEL
LIN {X 0,Y 587.471,Z 331.981,A -85,B 0,C 180,E1 -1609.488,E2 -1609.488} C_VEL
LIN {X 0,Y 587.421,Z 342.499,A -85,B 0,C 180,E1 -1610.184,E2 -1610.184} C_VEL
LIN {X 0,Y 587.348,Z 353.046,A -85,B 0,C 180,E1 -1611.051,E2 -1611.051} C_VEL
LIN {X 0,Y 587.3,Z 361.574,A -85,B 0,C 180,E1 -1611.917,E2 -1611.917} C_VEL
LIN {X 0,Y 587.248,Z 369.9,A -85,B 0,C 180,E1 -1612.954,E2 -1612.954} C_VEL
LIN {X 0,Y 587.218,Z 376.61,A -85,B 0,C 180,E1 -1613.989,E2 -1613.989} C_VEL
LIN {X 0,Y 587.146,Z 382.756,A -85,B 0,C 180,E1 -1615.194,E2 -1615.194} C_VEL
LIN {X 0,Y 587.213,Z 386.743,A -85,B 0,C 180,E1 -1616.226,E2 -1616.226} C_VEL
LIN {X 0,Y 587.131,Z 389.697,A -85,B 0,C 180,E1 -1617.256,E2 -1617.256} C_VEL
LIN {X 0,Y 587.141,Z 391.134,A -85,B 0,C 180,E1 -1617.942,E2 -1617.942} C_VEL
LIN {X 0,Y 587.14,Z 392.756,A -85,B 0,C 180,E1 -1619.314,E2 -1619.314} C_VEL
LIN {X 0,Y 587.137,Z 392.996,A -85,B 0,C 180,E1 -1620,E2 -1620} C_VEL
LIN {X 0,Y 587.148,Z 392.231,A -85,B 0,C 180,E1 -1621.372,E2 -1621.372} C_VEL
LIN {X 0,Y 587.141,Z 391.278,A -85,B 0,C 180,E1 -1622.058,E2 -1622.058} C_VEL
LIN {X 0,Y 587.132,Z 389.891,A -85,B 0,C 180,E1 -1622.744,E2 -1622.744} C_VEL
LIN {X 0,Y 587.213,Z 387.019,A -85,B 0,C 180,E1 -1623.774,E2 -1623.774} C_VEL
LIN {X 0,Y 587.147,Z 383.127,A -85,B 0,C 180,E1 -1624.806,E2 -1624.806} C_VEL
LIN {X 0,Y 587.23,Z 378.103,A -85,B 0,C 180,E1 -1625.839,E2 -1625.839} C_VEL
LIN {X 0,Y 587.245,Z 370.548,A -85,B 0,C 180,E1 -1627.046,E2 -1627.046} C_VEL
LIN {X 0,Y 587.286,Z 362.35,A -85,B 0,C 180,E1 -1628.083,E2 -1628.083} C_VEL
LIN {X 0,Y 587.338,Z 353.987,A -85,B 0,C 180,E1 -1628.949,E2 -1628.949} C_VEL
LIN {X 0,Y 587.415,Z 343.704,A -85,B 0,C 180,E1 -1629.816,E2 -1629.816} C_VEL
LIN {X 0,Y 587.458,Z 333.492,A -85,B 0,C 180,E1 -1630.512,E2 -1630.512} C_VEL
LIN {X 0,Y 587.531,Z 322.029,A -85,B 0,C 180,E1 -1631.134,E2 -1631.134} C_VEL
LIN {X 0,Y 587.578,Z 310.89,A -85,B 0,C 180,E1 -1631.603,E2 -1631.603} C_VEL
LIN {X 0,Y 587.703,Z 298.273,A -85,B 0,C 180,E1 -1631.992,E2 -1631.992} C_VEL
LIN {X 0,Y 587.509,Z 292.46,A -85,B 0,C 180,E1 -1632.128,E2 -1632.128} C_VEL
LIN {X 0,Y 587.124,Z 289.895,A -85,B 0,C 180,E1 -1632.201,E2 -1632.201} C_VEL
LIN {X 0,Y 587.112,Z 287.121,A -85,B 0,C 180,E1 -1634.425,E2 -1634.425} C_VEL
LIN {X 0,Y 586.403,Z 286.439,A -85,B 0,C 180,E1 -1634.994,E2 -1634.994} C_VEL
LIN {X 0,Y 583.518,Z 285.397,A -85,B 0,C 180,E1 -1635.918,E2 -1635.918} C_VEL
LIN {X 0,Y 581.113,Z 284.574,A -85,B 0,C 180,E1 -1636.661,E2 -1636.661} C_VEL
LIN {X 0,Y 580.097,Z 283.915,A -85,B 0,C 180,E1 -1637.235,E2 -1637.235} C_VEL
LIN {X 0,Y 580.022,Z 283.684,A -85,B 0,C 180,E1 -1637.429,E2 -1637.429} C_VEL
LIN {X 0,Y 580.044,Z 280.799,A -85,B 0,C 180,E1 -1639.832,E2 -1639.832} C_VEL
LIN {X 0,Y 580.033,Z 278.161,A -85,B 0,C 180,E1 -1642.062,E2 -1642.062} C_VEL
LIN {X 0,Y 580.049,Z 277.234,A -85,B 0,C 180,E1 -1642.951,E2 -1642.951} C_VEL
LIN {X 0,Y 580.251,Z 277.205,A -85,B 0,C 180,E1 -1645.082,E2 -1645.082} C_VEL
LIN {X 0,Y 580.295,Z 277.196,A -85,B 0,C 180,E1 -1647.857,E2 -1647.857} C_VEL
LIN {X 0,Y 580.279,Z 277.203,A -85,B 0,C 180,E1 -1650.693,E2 -1650.693} C_VEL
LIN {X 0,Y 580.287,Z 277.197,A -85,B 0,C 180,E1 -1653.313,E2 -1653.313} C_VEL
LIN {X 0,Y 580.248,Z 277.203,A -85,B 0,C 180,E1 -1655.756,E2 -1655.756} C_VEL
LIN {X 0,Y 580.292,Z 277.206,A -85,B 0,C 180,E1 -1658.146,E2 -1658.146} C_VEL
LIN {X 0,Y 580.302,Z 277.196,A -85,B 0,C 180,E1 -1660.843,E2 -1660.843} C_VEL
LIN {X 0,Y 580.283,Z 277.202,A -85,B 0,C 180,E1 -1663.658,E2 -1663.658} C_VEL
LIN {X 0,Y 580.281,Z 277.198,A -85,B 0,C 180,E1 -1666.609,E2 -1666.609} C_VEL
LIN {X 0,Y 580.301,Z 277.197,A -85,B 0,C 180,E1 -1669.157,E2 -1669.157} C_VEL
LIN {X 0,Y 580.292,Z 277.201,A -85,B 0,C 180,E1 -1671.927,E2 -1671.927} C_VEL
LIN {X 0,Y 580.253,Z 277.202,A -85,B 0,C 180,E1 -1674.453,E2 -1674.453} C_VEL
LIN {X 0,Y 580.211,Z 277.37,A -85,B 0,C 180,E1 -1675.704,E2 -1675.704} C_VEL
LIN {X 0,Y 580.176,Z 282.865,A -85,B 0,C 180,E1 -1678.608,E2 -1678.608} C_VEL
LIN {X 0,Y 580.1,Z 287.291,A -85,B 0,C 180,E1 -1681.013,E2 -1681.013} C_VEL
LIN {X 0,Y 580.145,Z 292.217,A -85,B 0,C 180,E1 -1683.696,E2 -1683.696} C_VEL
LIN {X 0,Y 580.129,Z 297.188,A -85,B 0,C 180,E1 -1686.435,E2 -1686.435} C_VEL
LIN {X 0,Y 580.131,Z 301.688,A -85,B 0,C 180,E1 -1688.879,E2 -1688.879} C_VEL
LIN {X 0,Y 580.097,Z 306.864,A -85,B 0,C 180,E1 -1691.639,E2 -1691.639} C_VEL
LIN {X 0,Y 580.075,Z 312.394,A -85,B 0,C 180,E1 -1694.541,E2 -1694.541} C_VEL
LIN {X 0,Y 580.053,Z 316.541,A -85,B 0,C 180,E1 -1696.691,E2 -1696.691} C_VEL
LIN {X 0,Y 580.069,Z 318.701,A -85,B 0,C 180,E1 -1697.737,E2 -1697.737} C_VEL
LIN {X 0,Y 580.79,Z 324.452,A -85,B 0,C 180,E1 -1697.863,E2 -1697.863} C_VEL
LIN {X 0,Y 580.672,Z 337.079,A -85,B 0,C 180,E1 -1698.215,E2 -1698.215} C_VEL
LIN {X 0,Y 580.579,Z 348.836,A -85,B 0,C 180,E1 -1698.673,E2 -1698.673} C_VEL
LIN {X 0,Y 580.509,Z 360.535,A -85,B 0,C 180,E1 -1699.272,E2 -1699.272} C_VEL
LIN {X 0,Y 580.418,Z 372.484,A -85,B 0,C 180,E1 -1700.064,E2 -1700.064} C_VEL
LIN {X 0,Y 580.333,Z 381.078,A -85,B 0,C 180,E1 -1700.766,E2 -1700.766} C_VEL
LIN {X 0,Y 580.264,Z 389.962,A -85,B 0,C 180,E1 -1701.643,E2 -1701.643} C_VEL
LIN {X 0,Y 580.2,Z 397.317,A -85,B 0,C 180,E1 -1702.518,E2 -1702.518} C_VEL
LIN {X 0,Y 580.135,Z 405.006,A -85,B 0,C 180,E1 -1703.637,E2 -1703.637} C_VEL
LIN {X 0,Y 580.086,Z 411.155,A -85,B 0,C 180,E1 -1704.787,E2 -1704.787} C_VEL
LIN {X 0,Y 580.105,Z 415.503,A -85,B 0,C 180,E1 -1705.831,E2 -1705.831} C_VEL
LIN {X 0,Y 580.123,Z 417.83,A -85,B 0,C 180,E1 -1706.527,E2 -1706.527} C_VEL
LIN {X 0,Y 580.043,Z 419.676,A -85,B 0,C 180,E1 -1707.222,E2 -1707.222} C_VEL
LIN {X 0,Y 580.046,Z 422.14,A -85,B 0,C 180,E1 -1708.611,E2 -1708.611} C_VEL
LIN {X 0,Y 580.041,Z 422.751,A -85,B 0,C 180,E1 -1709.306,E2 -1709.306} C_VEL
LIN {X 0,Y 580.04,Z 422.812,A -85,B 0,C 180,E1 -1710.694,E2 -1710.694} C_VEL
LIN {X 0,Y 580.047,Z 422.241,A -85,B 0,C 180,E1 -1711.389,E2 -1711.389} C_VEL
LIN {X 0,Y 580.044,Z 419.905,A -85,B 0,C 180,E1 -1712.778,E2 -1712.778} C_VEL
LIN {X 0,Y 580.11,Z 417.032,A -85,B 0,C 180,E1 -1713.821,E2 -1713.821} C_VEL
LIN {X 0,Y 580.053,Z 413.125,A -85,B 0,C 180,E1 -1714.865,E2 -1714.865} C_VEL
LIN {X 0,Y 580.163,Z 408.075,A -85,B 0,C 180,E1 -1715.91,E2 -1715.91} C_VEL
LIN {X 0,Y 580.157,Z 401.742,A -85,B 0,C 180,E1 -1716.958,E2 -1716.958} C_VEL
LIN {X 0,Y 580.241,Z 393.873,A -85,B 0,C 180,E1 -1718.007,E2 -1718.007} C_VEL
LIN {X 0,Y 580.308,Z 383.978,A -85,B 0,C 180,E1 -1719.058,E2 -1719.058} C_VEL
LIN {X 0,Y 580.389,Z 374.793,A -85,B 0,C 180,E1 -1719.848,E2 -1719.848} C_VEL
LIN {X 0,Y 580.46,Z 364.863,A -85,B 0,C 180,E1 -1720.552,E2 -1720.552} C_VEL
LIN {X 0,Y 580.549,Z 352.665,A -85,B 0,C 180,E1 -1721.24,E2 -1721.24} C_VEL
LIN {X 0,Y 580.661,Z 339.949,A -85,B 0,C 180,E1 -1721.777,E2 -1721.777} C_VEL
LIN {X 0,Y 580.739,Z 328.096,A -85,B 0,C 180,E1 -1722.138,E2 -1722.138} C_VEL
LIN {X 0,Y 580.663,Z 322.44,A -85,B 0,C 180,E1 -1722.273,E2 -1722.273} C_VEL
LIN {X 0,Y 580.085,Z 318.531,A -85,B 0,C 180,E1 -1722.374,E2 -1722.374} C_VEL
LIN {X 0,Y 580.102,Z 313.95,A -85,B 0,C 180,E1 -1724.739,E2 -1724.739} C_VEL
LIN {X 0,Y 580.056,Z 308.417,A -85,B 0,C 180,E1 -1727.632,E2 -1727.632} C_VEL
LIN {X 0,Y 580.1,Z 304.268,A -85,B 0,C 180,E1 -1729.83,E2 -1729.83} C_VEL
LIN {X 0,Y 580.128,Z 300.119,A -85,B 0,C 180,E1 -1732.059,E2 -1732.059} C_VEL
LIN {X 0,Y 580.155,Z 294.613,A -85,B 0,C 180,E1 -1735.087,E2 -1735.087} C_VEL
LIN {X 0,Y 580.151,Z 289.584,A -85,B 0,C 180,E1 -1737.83,E2 -1737.83} C_VEL
LIN {X 0,Y 580.18,Z 284.354,A -85,B 0,C 180,E1 -1740.677,E2 -1740.677} C_VEL
LIN {X 0,Y 580.19,Z 279.488,A -85,B 0,C 180,E1 -1743.299,E2 -1743.299} C_VEL
LIN {X 0,Y 580.264,Z 277.209,A -85,B 0,C 180,E1 -1744.553,E2 -1744.553} C_VEL
LIN {X 0,Y 580.29,Z 277.205,A -85,B 0,C 180,E1 -1747.269,E2 -1747.269} C_VEL
LIN {X 0,Y 580.296,Z 277.201,A -85,B 0,C 180,E1 -1750.271,E2 -1750.271} C_VEL
LIN {X 0,Y 580.282,Z 277.204,A -85,B 0,C 180,E1 -1752.706,E2 -1752.706} C_VEL
LIN {X 0,Y 580.258,Z 277.206,A -85,B 0,C 180,E1 -1755.611,E2 -1755.611} C_VEL
LIN {X 0,Y 580.28,Z 277.203,A -85,B 0,C 180,E1 -1758.231,E2 -1758.231} C_VEL
LIN {X 0,Y 580.287,Z 277.202,A -85,B 0,C 180,E1 -1760.966,E2 -1760.966} C_VEL
LIN {X 0,Y 580.253,Z 277.207,A -85,B 0,C 180,E1 -1763.595,E2 -1763.595} C_VEL
LIN {X 0,Y 580.21,Z 277.299,A -85,B 0,C 180,E1 -1765.705,E2 -1765.705} C_VEL
LIN {X 0,Y 580.164,Z 282.803,A -85,B 0,C 180,E1 -1768.608,E2 -1768.608} C_VEL
LIN {X 0,Y 580.127,Z 287.364,A -85,B 0,C 180,E1 -1771.015,E2 -1771.015} C_VEL
LIN {X 0,Y 580.145,Z 292.186,A -85,B 0,C 180,E1 -1773.696,E2 -1773.696} C_VEL
LIN {X 0,Y 580.129,Z 297.188,A -85,B 0,C 180,E1 -1776.435,E2 -1776.435} C_VEL
LIN {X 0,Y 580.131,Z 301.688,A -85,B 0,C 180,E1 -1778.879,E2 -1778.879} C_VEL
LIN {X 0,Y 580.097,Z 306.864,A -85,B 0,C 180,E1 -1781.639,E2 -1781.639} C_VEL
LIN {X 0,Y 580.075,Z 312.394,A -85,B 0,C 180,E1 -1784.541,E2 -1784.541} C_VEL
LIN {X 0,Y 580.053,Z 316.541,A -85,B 0,C 180,E1 -1786.691,E2 -1786.691} C_VEL
LIN {X 0,Y 580.072,Z 318.751,A -85,B 0,C 180,E1 -1787.737,E2 -1787.737} C_VEL
LIN {X 0,Y 580.79,Z 324.407,A -85,B 0,C 180,E1 -1787.863,E2 -1787.863} C_VEL
LIN {X 0,Y 580.698,Z 335.904,A -85,B 0,C 180,E1 -1788.175,E2 -1788.175} C_VEL
LIN {X 0,Y 580.614,Z 347.164,A -85,B 0,C 180,E1 -1788.597,E2 -1788.597} C_VEL
LIN {X 0,Y 580.509,Z 360.549,A -85,B 0,C 180,E1 -1789.272,E2 -1789.272} C_VEL
LIN {X 0,Y 580.433,Z 371.276,A -85,B 0,C 180,E1 -1789.976,E2 -1789.976} C_VEL
LIN {X 0,Y 580.333,Z 381.074,A -85,B 0,C 180,E1 -1790.766,E2 -1790.766} C_VEL
LIN {X 0,Y 580.264,Z 389.991,A -85,B 0,C 180,E1 -1791.643,E2 -1791.643} C_VEL
LIN {X 0,Y 580.206,Z 398.677,A -85,B 0,C 180,E1 -1792.693,E2 -1792.693} C_VEL
LIN {X 0,Y 580.137,Z 405.595,A -85,B 0,C 180,E1 -1793.741,E2 -1793.741} C_VEL
LIN {X 0,Y 580.085,Z 411.136,A -85,B 0,C 180,E1 -1794.787,E2 -1794.787} C_VEL
LIN {X 0,Y 580.105,Z 415.493,A -85,B 0,C 180,E1 -1795.831,E2 -1795.831} C_VEL
LIN {X 0,Y 580.123,Z 417.828,A -85,B 0,C 180,E1 -1796.527,E2 -1796.527} C_VEL
LIN {X 0,Y 580.043,Z 419.688,A -85,B 0,C 180,E1 -1797.222,E2 -1797.222} C_VEL
LIN {X 0,Y 580.046,Z 422.134,A -85,B 0,C 180,E1 -1798.611,E2 -1798.611} C_VEL
LIN {X 0,Y 580.041,Z 422.757,A -85,B 0,C 180,E1 -1799.306,E2 -1799.306} C_VEL
LIN {X 0,Y 580.04,Z 422.807,A -85,B 0,C 180,E1 -1800.694,E2 -1800.694} C_VEL
LIN {X 0,Y 580.047,Z 422.242,A -85,B 0,C 180,E1 -1801.389,E2 -1801.389} C_VEL
LIN {X 0,Y 580.044,Z 419.902,A -85,B 0,C 180,E1 -1802.778,E2 -1802.778} C_VEL
LIN {X 0,Y 580.11,Z 417.031,A -85,B 0,C 180,E1 -1803.821,E2 -1803.821} C_VEL
LIN {X 0,Y 580.053,Z 413.126,A -85,B 0,C 180,E1 -1804.865,E2 -1804.865} C_VEL
LIN {X 0,Y 580.163,Z 408.077,A -85,B 0,C 180,E1 -1805.91,E2 -1805.91} C_VEL
LIN {X 0,Y 580.157,Z 401.738,A -85,B 0,C 180,E1 -1806.958,E2 -1806.958} C_VEL
LIN {X 0,Y 580.241,Z 393.872,A -85,B 0,C 180,E1 -1808.007,E2 -1808.007} C_VEL
LIN {X 0,Y 580.299,Z 383.997,A -85,B 0,C 180,E1 -1809.059,E2 -1809.059} C_VEL
LIN {X 0,Y 580.389,Z 374.796,A -85,B 0,C 180,E1 -1809.848,E2 -1809.848} C_VEL
LIN {X 0,Y 580.46,Z 364.838,A -85,B 0,C 180,E1 -1810.552,E2 -1810.552} C_VEL
LIN {X 0,Y 580.522,Z 354.052,A -85,B 0,C 180,E1 -1811.169,E2 -1811.169} C_VEL
LIN {X 0,Y 580.642,Z 341.02,A -85,B 0,C 180,E1 -1811.741,E2 -1811.741} C_VEL
LIN {X 0,Y 580.742,Z 328.102,A -85,B 0,C 180,E1 -1812.138,E2 -1812.138} C_VEL
LIN {X 0,Y 580.653,Z 322.169,A -85,B 0,C 180,E1 -1812.279,E2 -1812.279} C_VEL
LIN {X 0,Y 580.085,Z 318.531,A -85,B 0,C 180,E1 -1812.374,E2 -1812.374} C_VEL
LIN {X 0,Y 580.102,Z 313.95,A -85,B 0,C 180,E1 -1814.739,E2 -1814.739} C_VEL
LIN {X 0,Y 580.056,Z 308.418,A -85,B 0,C 180,E1 -1817.632,E2 -1817.632} C_VEL
